LIN {X 0,Y 369.044,Z 241.011,A -85,B 0,C 180,E1 -12789.865,E2 -12789.865} C_VEL
LIN {X 0,Y 369.022,Z 241.014,A -85,B 0,C 180,E1 -12793.768,E2 -12793.768} C_VEL
LIN {X 0,Y 368.974,Z 241.02,A -85,B 0,C 180,E1 -12797.739,E2 -12797.739} C_VEL
LIN {X 0,Y 368.891,Z 241.032,A -85,B 0,C 180,E1 -12801.217,E2 -12801.217} C_VEL
LIN {X 0,Y 368.912,Z 241.029,A -85,B 0,C 180,E1 -12804.774,E2 -12804.774} C_VEL
LIN {X 0,Y 368.894,Z 241.025,A -85,B 0,C 180,E1 -12808.438,E2 -12808.438} C_VEL
LIN {X 0,Y 368.874,Z 241.03,A -85,B 0,C 180,E1 -12812.235,E2 -12812.235} C_VEL
LIN {X 0,Y 368.905,Z 241.028,A -85,B 0,C 180,E1 -12814.998,E2 -12814.998} C_VEL
LIN {X 0,Y 368.887,Z 241.036,A -85,B 0,C 180,E1 -12818.638,E2 -12818.638} C_VEL
LIN {X 0,Y 368.952,Z 241.097,A -85,B 0,C 180,E1 -12820.366,E2 -12820.366} C_VEL
LIN {X 0,Y 370.279,Z 247.105,A -85,B 0,C 180,E1 -12822.072,E2 -12822.072} C_VEL
LIN {X 0,Y 372.182,Z 257.131,A -85,B 0,C 180,E1 -12824.693,E2 -12824.693} C_VEL
LIN {X 0,Y 372.185,Z 259.385,A -85,B 0,C 180,E1 -12825.156,E2 -12825.156} C_VEL
LIN {X 0,Y 376.972,Z 282.842,A -85,B 0,C 180,E1 -12825.983,E2 -12825.983} C_VEL
LIN {X 0,Y 377.58,Z 287.336,A -85,B 0,C 180,E1 -12826.115,E2 -12826.115} C_VEL
LIN {X 0,Y 376.049,Z 367.06,A -85,B 0,C 180,E1 -12827.695,E2 -12827.695} C_VEL
LIN {X 0,Y 375.45,Z 380.427,A -85,B 0,C 180,E1 -12828.176,E2 -12828.176} C_VEL
LIN {X 0,Y 374.723,Z 393.48,A -85,B 0,C 180,E1 -12828.884,E2 -12828.884} C_VEL
LIN {X 0,Y 373.829,Z 405.095,A -85,B 0,C 180,E1 -12829.742,E2 -12829.742} C_VEL
LIN {X 0,Y 372.648,Z 417.198,A -85,B 0,C 180,E1 -12830.894,E2 -12830.894} C_VEL
LIN {X 0,Y 371.644,Z 427.056,A -85,B 0,C 180,E1 -12832.08,E2 -12832.08} C_VEL
LIN {X 0,Y 370.718,Z 435.571,A -85,B 0,C 180,E1 -12833.334,E2 -12833.334} C_VEL
LIN {X 0,Y 369.704,Z 444.74,A -85,B 0,C 180,E1 -12835.006,E2 -12835.006} C_VEL
LIN {X 0,Y 368.986,Z 451.255,A -85,B 0,C 180,E1 -12836.473,E2 -12836.473} C_VEL
LIN {X 0,Y 368.284,Z 457.921,A -85,B 0,C 180,E1 -12838.348,E2 -12838.348} C_VEL
LIN {X 0,Y 367.826,Z 462.929,A -85,B 0,C 180,E1 -12840.214,E2 -12840.214} C_VEL
LIN {X 0,Y 367.579,Z 465.737,A -85,B 0,C 180,E1 -12841.571,E2 -12841.571} C_VEL
LIN {X 0,Y 367.38,Z 467.49,A -85,B 0,C 180,E1 -12842.671,E2 -12842.671} C_VEL
LIN {X 0,Y 367.234,Z 469.127,A -85,B 0,C 180,E1 -12844.076,E2 -12844.076} C_VEL
LIN {X 0,Y 367.144,Z 469.909,A -85,B 0,C 180,E1 -12845.095,E2 -12845.095} C_VEL
LIN {X 0,Y 367.118,Z 470.416,A -85,B 0,C 180,E1 -12846.752,E2 -12846.752} C_VEL
LIN {X 0,Y 367.121,Z 469.889,A -85,B 0,C 180,E1 -12848.672,E2 -12848.672} C_VEL
LIN {X 0,Y 367.223,Z 468.929,A -85,B 0,C 180,E1 -12849.851,E2 -12849.851} C_VEL
LIN {X 0,Y 367.326,Z 467.538,A -85,B 0,C 180,E1 -12851.02,E2 -12851.02} C_VEL
LIN {X 0,Y 367.596,Z 464.278,A -85,B 0,C 180,E1 -12852.91,E2 -12852.91} C_VEL
LIN {X 0,Y 367.867,Z 460.491,A -85,B 0,C 180,E1 -12854.488,E2 -12854.488} C_VEL
LIN {X 0,Y 368.367,Z 455.285,A -85,B 0,C 180,E1 -12856.176,E2 -12856.176} C_VEL
LIN {X 0,Y 368.997,Z 448.471,A -85,B 0,C 180,E1 -12857.908,E2 -12857.908} C_VEL
LIN {X 0,Y 369.827,Z 440.094,A -85,B 0,C 180,E1 -12859.6,E2 -12859.6} C_VEL
LIN {X 0,Y 370.758,Z 430.811,A -85,B 0,C 180,E1 -12861.106,E2 -12861.106} C_VEL
LIN {X 0,Y 371.714,Z 420.895,A -85,B 0,C 180,E1 -12862.396,E2 -12862.396} C_VEL
LIN {X 0,Y 372.696,Z 410.311,A -85,B 0,C 180,E1 -12863.504,E2 -12863.504} C_VEL
LIN {X 0,Y 373.641,Z 398.688,A -85,B 0,C 180,E1 -12864.469,E2 -12864.469} C_VEL
LIN {X 0,Y 374.319,Z 386.768,A -85,B 0,C 180,E1 -12865.222,E2 -12865.222} C_VEL
LIN {X 0,Y 375.026,Z 373.695,A -85,B 0,C 180,E1 -12865.803,E2 -12865.803} C_VEL
LIN {X 0,Y 375.431,Z 360.14,A -85,B 0,C 180,E1 -12866.177,E2 -12866.177} C_VEL
LIN {X 0,Y 376.575,Z 285.809,A -85,B 0,C 180,E1 -12867.62,E2 -12867.62} C_VEL
LIN {X 0,Y 371.712,Z 259.806,A -85,B 0,C 180,E1 -12868.444,E2 -12868.444} C_VEL
LIN {X 0,Y 371.685,Z 258.504,A -85,B 0,C 180,E1 -12868.647,E2 -12868.647} C_VEL
LIN {X 0,Y 371.677,Z 254.292,A -85,B 0,C 180,E1 -12869.73,E2 -12869.73} C_VEL
LIN {X 0,Y 370.534,Z 247.731,A -85,B 0,C 180,E1 -12871.523,E2 -12871.523} C_VEL
LIN {X 0,Y 369.47,Z 246.002,A -85,B 0,C 180,E1 -12872.056,E2 -12872.056} C_VEL
LIN {X 0,Y 366.012,Z 243.763,A -85,B 0,C 180,E1 -12872.906,E2 -12872.906} C_VEL
LIN {X 0,Y 362.72,Z 242.239,A -85,B 0,C 180,E1 -12873.814,E2 -12873.814} C_VEL
LIN {X 0,Y 361.924,Z 241.9,A -85,B 0,C 180,E1 -12874.431,E2 -12874.431} C_VEL
LIN {X 0,Y 362.127,Z 241.873,A -85,B 0,C 180,E1 -12876.688,E2 -12876.688} C_VEL
LIN {X 0,Y 361.999,Z 241.891,A -85,B 0,C 180,E1 -12880.064,E2 -12880.064} C_VEL
LIN {X 0,Y 361.965,Z 241.895,A -85,B 0,C 180,E1 -12883.901,E2 -12883.901} C_VEL
LIN {X 0,Y 361.935,Z 241.904,A -85,B 0,C 180,E1 -12887.941,E2 -12887.941} C_VEL
LIN {X 0,Y 361.823,Z 241.914,A -85,B 0,C 180,E1 -12891.658,E2 -12891.658} C_VEL
LIN {X 0,Y 361.858,Z 241.905,A -85,B 0,C 180,E1 -12895.296,E2 -12895.296} C_VEL
LIN {X 0,Y 361.827,Z 241.901,A -85,B 0,C 180,E1 -12899.077,E2 -12899.077} C_VEL
LIN {X 0,Y 361.819,Z 241.911,A -85,B 0,C 180,E1 -12902.949,E2 -12902.949} C_VEL
LIN {X 0,Y 361.837,Z 241.897,A -85,B 0,C 180,E1 -12905.641,E2 -12905.641} C_VEL
LIN {X 0,Y 361.8,Z 241.916,A -85,B 0,C 180,E1 -12909.021,E2 -12909.021} C_VEL
LIN {X 0,Y 361.806,Z 241.902,A -85,B 0,C 180,E1 -12912.834,E2 -12912.834} C_VEL
LIN {X 0,Y 361.792,Z 241.915,A -85,B 0,C 180,E1 -12915.952,E2 -12915.952} C_VEL
LIN {X 0,Y 361.791,Z 241.907,A -85,B 0,C 180,E1 -12919.254,E2 -12919.254} C_VEL
LIN {X 0,Y 361.845,Z 241.898,A -85,B 0,C 180,E1 -12922.986,E2 -12922.986} C_VEL
LIN {X 0,Y 361.843,Z 241.911,A -85,B 0,C 180,E1 -12926.636,E2 -12926.636} C_VEL
LIN {X 0,Y 361.834,Z 241.894,A -85,B 0,C 180,E1 -12929.674,E2 -12929.674} C_VEL
LIN {X 0,Y 361.844,Z 241.899,A -85,B 0,C 180,E1 -12933.472,E2 -12933.472} C_VEL
LIN {X 0,Y 361.865,Z 241.909,A -85,B 0,C 180,E1 -12937.148,E2 -12937.148} C_VEL
LIN {X 0,Y 361.897,Z 241.888,A -85,B 0,C 180,E1 -12940.728,E2 -12940.728} C_VEL
LIN {X 0,Y 361.938,Z 241.884,A -85,B 0,C 180,E1 -12944.23,E2 -12944.23} C_VEL
LIN {X 0,Y 361.995,Z 241.887,A -85,B 0,C 180,E1 -12946.532,E2 -12946.532} C_VEL
LIN {X 0,Y 361.993,Z 241.889,A -85,B 0,C 180,E1 -12949.941,E2 -12949.941} C_VEL
LIN {X 0,Y 362.118,Z 241.853,A -85,B 0,C 180,E1 -12953.317,E2 -12953.317} C_VEL
LIN {X 0,Y 362.266,Z 241.852,A -85,B 0,C 180,E1 -12957.78,E2 -12957.78} C_VEL
LIN {X 0,Y 362.202,Z 241.861,A -85,B 0,C 180,E1 -12961.116,E2 -12961.116} C_VEL
LIN {X 0,Y 362.261,Z 241.852,A -85,B 0,C 180,E1 -12962.227,E2 -12962.227} C_VEL
LIN {X 0,Y 362.145,Z 241.857,A -85,B 0,C 180,E1 -12966.69,E2 -12966.69} C_VEL
LIN {X 0,Y 362.004,Z 241.89,A -85,B 0,C 180,E1 -12970.066,E2 -12970.066} C_VEL
LIN {X 0,Y 362.006,Z 241.879,A -85,B 0,C 180,E1 -12973.902,E2 -12973.902} C_VEL
LIN {X 0,Y 361.936,Z 241.889,A -85,B 0,C 180,E1 -12976.937,E2 -12976.937} C_VEL
LIN {X 0,Y 361.896,Z 241.906,A -85,B 0,C 180,E1 -12980.464,E2 -12980.464} C_VEL
LIN {X 0,Y 361.904,Z 241.882,A -85,B 0,C 180,E1 -12984.115,E2 -12984.115} C_VEL
LIN {X 0,Y 361.853,Z 241.909,A -85,B 0,C 180,E1 -12987.787,E2 -12987.787} C_VEL
LIN {X 0,Y 361.858,Z 241.899,A -85,B 0,C 180,E1 -12991.287,E2 -12991.287} C_VEL
LIN {X 0,Y 361.865,Z 241.907,A -85,B 0,C 180,E1 -12994.282,E2 -12994.282} C_VEL
LIN {X 0,Y 361.871,Z 241.901,A -85,B 0,C 180,E1 -12997.224,E2 -12997.224} C_VEL
LIN {X 0,Y 361.825,Z 241.912,A -85,B 0,C 180,E1 -13000.752,E2 -13000.752} C_VEL
LIN {X 0,Y 361.826,Z 241.913,A -85,B 0,C 180,E1 -13004.37,E2 -13004.37} C_VEL
LIN {X 0,Y 361.842,Z 241.912,A -85,B 0,C 180,E1 -13007.571,E2 -13007.571} C_VEL
LIN {X 0,Y 361.855,Z 241.911,A -85,B 0,C 180,E1 -13011.573,E2 -13011.573} C_VEL
LIN {X 0,Y 361.887,Z 241.907,A -85,B 0,C 180,E1 -13014.656,E2 -13014.656} C_VEL
LIN {X 0,Y 361.851,Z 241.913,A -85,B 0,C 180,E1 -13018.371,E2 -13018.371} C_VEL
LIN {X 0,Y 361.94,Z 241.978,A -85,B 0,C 180,E1 -13021.196,E2 -13021.196} C_VEL
LIN {X 0,Y 363.7,Z 250.571,A -85,B 0,C 180,E1 -13023.611,E2 -13023.611} C_VEL
LIN {X 0,Y 365.297,Z 259.104,A -85,B 0,C 180,E1 -13025.868,E2 -13025.868} C_VEL
LIN {X 0,Y 364.796,Z 266.345,A -85,B 0,C 180,E1 -13027.635,E2 -13027.635} C_VEL
LIN {X 0,Y 364.608,Z 268.699,A -85,B 0,C 180,E1 -13028.152,E2 -13028.152} C_VEL
LIN {X 0,Y 365.93,Z 276.421,A -85,B 0,C 180,E1 -13028.437,E2 -13028.437} C_VEL
LIN {X 0,Y 369.774,Z 299.232,A -85,B 0,C 180,E1 -13029.125,E2 -13029.125} C_VEL
LIN {X 0,Y 368.476,Z 376.627,A -85,B 0,C 180,E1 -13030.682,E2 -13030.682} C_VEL
LIN {X 0,Y 367.861,Z 389.768,A -85,B 0,C 180,E1 -13031.155,E2 -13031.155} C_VEL
LIN {X 0,Y 367.089,Z 401.886,A -85,B 0,C 180,E1 -13031.801,E2 -13031.801} C_VEL
LIN {X 0,Y 366.077,Z 414.134,A -85,B 0,C 180,E1 -13032.687,E2 -13032.687} C_VEL
LIN {X 0,Y 365.009,Z 425.73,A -85,B 0,C 180,E1 -13033.787,E2 -13033.787} C_VEL
LIN {X 0,Y 364.045,Z 436.165,A -85,B 0,C 180,E1 -13035.034,E2 -13035.034} C_VEL
LIN {X 0,Y 363.234,Z 444.713,A -85,B 0,C 180,E1 -13036.289,E2 -13036.289} C_VEL
LIN {X 0,Y 362.169,Z 453.947,A -85,B 0,C 180,E1 -13037.958,E2 -13037.958} C_VEL
LIN {X 0,Y 361.457,Z 461.37,A -85,B 0,C 180,E1 -13039.638,E2 -13039.638} C_VEL
LIN {X 0,Y 360.855,Z 468.19,A -85,B 0,C 180,E1 -13041.6,E2 -13041.6} C_VEL
LIN {X 0,Y 360.52,Z 472.681,A -85,B 0,C 180,E1 -13043.282,E2 -13043.282} C_VEL
LIN {X 0,Y 360.409,Z 475.047,A -85,B 0,C 180,E1 -13044.404,E2 -13044.404} C_VEL
LIN {X 0,Y 360.355,Z 476.982,A -85,B 0,C 180,E1 -13045.525,E2 -13045.525} C_VEL
LIN {X 0,Y 360.279,Z 478.488,A -85,B 0,C 180,E1 -13046.644,E2 -13046.644} C_VEL
LIN {X 0,Y 360.254,Z 480.203,A -85,B 0,C 180,E1 -13048.881,E2 -13048.881} C_VEL
LIN {X 0,Y 360.28,Z 480.477,A -85,B 0,C 180,E1 -13049.999,E2 -13049.999} C_VEL
LIN {X 0,Y 360.253,Z 480.354,A -85,B 0,C 180,E1 -13051.117,E2 -13051.117} C_VEL
LIN {X 0,Y 360.282,Z 478.849,A -85,B 0,C 180,E1 -13053.354,E2 -13053.354} C_VEL
LIN {X 0,Y 360.383,Z 477.507,A -85,B 0,C 180,E1 -13054.473,E2 -13054.473} C_VEL
LIN {X 0,Y 360.47,Z 474.804,A -85,B 0,C 180,E1 -13056.084,E2 -13056.084} C_VEL
LIN {X 0,Y 360.757,Z 470.803,A -85,B 0,C 180,E1 -13057.837,E2 -13057.837} C_VEL
LIN {X 0,Y 361.229,Z 465.814,A -85,B 0,C 180,E1 -13059.518,E2 -13059.518} C_VEL
LIN {X 0,Y 361.887,Z 459.549,A -85,B 0,C 180,E1 -13061.197,E2 -13061.197} C_VEL
LIN {X 0,Y 362.802,Z 451.718,A -85,B 0,C 180,E1 -13062.871,E2 -13062.871} C_VEL
LIN {X 0,Y 363.967,Z 441.947,A -85,B 0,C 180,E1 -13064.537,E2 -13064.537} C_VEL
LIN {X 0,Y 364.975,Z 431.82,A -85,B 0,C 180,E1 -13065.925,E2 -13065.925} C_VEL
LIN {X 0,Y 366.099,Z 421.791,A -85,B 0,C 180,E1 -13067.022,E2 -13067.022} C_VEL
LIN {X 0,Y 367.139,Z 410.901,A -85,B 0,C 180,E1 -13067.978,E2 -13067.978} C_VEL
LIN {X 0,Y 368.134,Z 398.889,A -85,B 0,C 180,E1 -13068.792,E2 -13068.792} C_VEL
LIN {X 0,Y 368.934,Z 386.604,A -85,B 0,C 180,E1 -13069.4,E2 -13069.4} C_VEL
LIN {X 0,Y 369.469,Z 374.043,A -85,B 0,C 180,E1 -13069.804,E2 -13069.804} C_VEL
LIN {X 0,Y 370.794,Z 299.844,A -85,B 0,C 180,E1 -13071.297,E2 -13071.297} C_VEL
LIN {X 0,Y 366.754,Z 276.745,A -85,B 0,C 180,E1 -13072.058,E2 -13072.058} C_VEL
LIN {X 0,Y 365.053,Z 268.304,A -85,B 0,C 180,E1 -13072.397,E2 -13072.397} C_VEL
LIN {X 0,Y 365.707,Z 260.961,A -85,B 0,C 180,E1 -13074.101,E2 -13074.101} C_VEL
LIN {X 0,Y 363.888,Z 250.827,A -85,B 0,C 180,E1 -13076.78,E2 -13076.78} C_VEL
LIN {X 0,Y 361.943,Z 242.234,A -85,B 0,C 180,E1 -13079.183,E2 -13079.183} C_VEL
LIN {X 0,Y 361.888,Z 241.905,A -85,B 0,C 180,E1 -13079.682,E2 -13079.682} C_VEL
LIN {X 0,Y 361.865,Z 241.908,A -85,B 0,C 180,E1 -13083.367,E2 -13083.367} C_VEL
LIN {X 0,Y 361.869,Z 241.902,A -85,B 0,C 180,E1 -13087.016,E2 -13087.016} C_VEL
LIN {X 0,Y 361.818,Z 241.908,A -85,B 0,C 180,E1 -13090.749,E2 -13090.749} C_VEL
LIN {X 0,Y 361.821,Z 241.918,A -85,B 0,C 180,E1 -13094.366,E2 -13094.366} C_VEL
LIN {X 0,Y 361.834,Z 241.912,A -85,B 0,C 180,E1 -13097.567,E2 -13097.567} C_VEL
LIN {X 0,Y 361.845,Z 241.905,A -85,B 0,C 180,E1 -13101.569,E2 -13101.569} C_VEL
LIN {X 0,Y 361.872,Z 241.905,A -85,B 0,C 180,E1 -13104.653,E2 -13104.653} C_VEL
LIN {X 0,Y 361.839,Z 241.908,A -85,B 0,C 180,E1 -13108.367,E2 -13108.367} C_VEL
LIN {X 0,Y 361.867,Z 241.909,A -85,B 0,C 180,E1 -13110.949,E2 -13110.949} C_VEL
LIN {X 0,Y 361.879,Z 241.909,A -85,B 0,C 180,E1 -13114.703,E2 -13114.703} C_VEL
LIN {X 0,Y 361.859,Z 241.905,A -85,B 0,C 180,E1 -13118.342,E2 -13118.342} C_VEL
LIN {X 0,Y 361.918,Z 241.892,A -85,B 0,C 180,E1 -13122.081,E2 -13122.081} C_VEL
LIN {X 0,Y 361.958,Z 241.893,A -85,B 0,C 180,E1 -13125.376,E2 -13125.376} C_VEL
LIN {X 0,Y 361.962,Z 241.896,A -85,B 0,C 180,E1 -13128.801,E2 -13128.801} C_VEL
LIN {X 0,Y 362.08,Z 241.876,A -85,B 0,C 180,E1 -13132.187,E2 -13132.187} C_VEL
LIN {X 0,Y 362.092,Z 241.879,A -85,B 0,C 180,E1 -13134.427,E2 -13134.427} C_VEL
LIN {X 0,Y 362.248,Z 241.861,A -85,B 0,C 180,E1 -13137.773,E2 -13137.773} C_VEL
LIN {X 0,Y 362.245,Z 241.86,A -85,B 0,C 180,E1 -13142.22,E2 -13142.22} C_VEL
LIN {X 0,Y 362.103,Z 241.876,A -85,B 0,C 180,E1 -13146.683,E2 -13146.683} C_VEL
LIN {X 0,Y 361.981,Z 241.891,A -85,B 0,C 180,E1 -13150.059,E2 -13150.059} C_VEL
LIN {X 0,Y 361.983,Z 241.891,A -85,B 0,C 180,E1 -13153.895,E2 -13153.895} C_VEL
LIN {X 0,Y 361.911,Z 241.897,A -85,B 0,C 180,E1 -13156.93,E2 -13156.93} C_VEL
LIN {X 0,Y 361.868,Z 241.908,A -85,B 0,C 180,E1 -13160.457,E2 -13160.457} C_VEL
LIN {X 0,Y 361.874,Z 241.91,A -85,B 0,C 180,E1 -13164.109,E2 -13164.109} C_VEL
LIN {X 0,Y 361.826,Z 241.911,A -85,B 0,C 180,E1 -13167.781,E2 -13167.781} C_VEL
LIN {X 0,Y 361.824,Z 241.912,A -85,B 0,C 180,E1 -13171.282,E2 -13171.282} C_VEL
LIN {X 0,Y 361.83,Z 241.914,A -85,B 0,C 180,E1 -13174.277,E2 -13174.277} C_VEL
LIN {X 0,Y 361.84,Z 241.909,A -85,B 0,C 180,E1 -13177.22,E2 -13177.22} C_VEL
LIN {X 0,Y 361.887,Z 242.014,A -85,B 0,C 180,E1 -13179.991,E2 -13179.991} C_VEL
LIN {X 0,Y 364.059,Z 252.05,A -85,B 0,C 180,E1 -13182.815,E2 -13182.815} C_VEL
LIN {X 0,Y 365.336,Z 259.235,A -85,B 0,C 180,E1 -13184.666,E2 -13184.666} C_VEL
LIN {X 0,Y 367.968,Z 271.225,A -85,B 0,C 180,E1 -13185.148,E2 -13185.148} C_VEL
LIN {X 0,Y 371.016,Z 287.413,A -85,B 0,C 180,E1 -13185.696,E2 -13185.696} C_VEL
LIN {X 0,Y 369.417,Z 367.303,A -85,B 0,C 180,E1 -13187.311,E2 -13187.311} C_VEL
LIN {X 0,Y 368.798,Z 380.614,A -85,B 0,C 180,E1 -13187.801,E2 -13187.801} C_VEL
LIN {X 0,Y 368.035,Z 393.611,A -85,B 0,C 180,E1 -13188.519,E2 -13188.519} C_VEL
LIN {X 0,Y 367.098,Z 405.197,A -85,B 0,C 180,E1 -13189.39,E2 -13189.39} C_VEL
LIN {X 0,Y 365.995,Z 416.282,A -85,B 0,C 180,E1 -13190.456,E2 -13190.456} C_VEL
LIN {X 0,Y 364.811,Z 427.131,A -85,B 0,C 180,E1 -13191.767,E2 -13191.767} C_VEL
LIN {X 0,Y 363.731,Z 436.589,A -85,B 0,C 180,E1 -13193.205,E2 -13193.205} C_VEL
LIN {X 0,Y 362.748,Z 445.105,A -85,B 0,C 180,E1 -13194.805,E2 -13194.805} C_VEL
LIN {X 0,Y 362.014,Z 451.36,A -85,B 0,C 180,E1 -13196.245,E2 -13196.245} C_VEL
LIN {X 0,Y 361.421,Z 456.486,A -85,B 0,C 180,E1 -13197.674,E2 -13197.674} C_VEL
LIN {X 0,Y 360.904,Z 461.912,A -85,B 0,C 180,E1 -13199.583,E2 -13199.583} C_VEL
LIN {X 0,Y 360.531,Z 465.562,A -85,B 0,C 180,E1 -13201.295,E2 -13201.295} C_VEL
LIN {X 0,Y 360.212,Z 468.571,A -85,B 0,C 180,E1 -13203.338,E2 -13203.338} C_VEL
LIN {X 0,Y 360.091,Z 469.685,A -85,B 0,C 180,E1 -13204.573,E2 -13204.573} C_VEL
LIN {X 0,Y 360.012,Z 470.491,A -85,B 0,C 180,E1 -13206.551,E2 -13206.551} C_VEL
LIN {X 0,Y 360.028,Z 470.193,A -85,B 0,C 180,E1 -13208.23,E2 -13208.23} C_VEL
LIN {X 0,Y 360.1,Z 469.392,A -85,B 0,C 180,E1 -13209.506,E2 -13209.506} C_VEL
LIN {X 0,Y 360.201,Z 468.215,A -85,B 0,C 180,E1 -13210.63,E2 -13210.63} C_VEL
LIN {X 0,Y 360.482,Z 464.784,A -85,B 0,C 180,E1 -13212.787,E2 -13212.787} C_VEL
LIN {X 0,Y 360.852,Z 460.199,A -85,B 0,C 180,E1 -13214.757,E2 -13214.757} C_VEL
LIN {X 0,Y 361.381,Z 454.762,A -85,B 0,C 180,E1 -13216.505,E2 -13216.505} C_VEL
LIN {X 0,Y 362.03,Z 447.928,A -85,B 0,C 180,E1 -13218.24,E2 -13218.24} C_VEL
LIN {X 0,Y 362.962,Z 439.404,A -85,B 0,C 180,E1 -13219.965,E2 -13219.965} C_VEL
LIN {X 0,Y 363.867,Z 430.631,A -85,B 0,C 180,E1 -13221.392,E2 -13221.392} C_VEL
LIN {X 0,Y 364.97,Z 419.749,A -85,B 0,C 180,E1 -13222.811,E2 -13222.811} C_VEL
LIN {X 0,Y 366,Z 408.903,A -85,B 0,C 180,E1 -13223.939,E2 -13223.939} C_VEL
LIN {X 0,Y 366.903,Z 397.811,A -85,B 0,C 180,E1 -13224.846,E2 -13224.846} C_VEL
LIN {X 0,Y 367.615,Z 385.485,A -85,B 0,C 180,E1 -13225.615,E2 -13225.615} C_VEL
LIN {X 0,Y 368.272,Z 372.83,A -85,B 0,C 180,E1 -13226.171,E2 -13226.171} C_VEL
LIN {X 0,Y 368.693,Z 360.056,A -85,B 0,C 180,E1 -13226.518,E2 -13226.518} C_VEL
LIN {X 0,Y 369.847,Z 286.54,A -85,B 0,C 180,E1 -13227.973,E2 -13227.973} C_VEL
LIN {X 0,Y 364.875,Z 260.049,A -85,B 0,C 180,E1 -13228.829,E2 -13228.829} C_VEL
LIN {X 0,Y 364.799,Z 258.971,A -85,B 0,C 180,E1 -13228.966,E2 -13228.966} C_VEL
LIN {X 0,Y 364.641,Z 255.007,A -85,B 0,C 180,E1 -13230.001,E2 -13230.001} C_VEL
LIN {X 0,Y 362.806,Z 245.13,A -85,B 0,C 180,E1 -13232.777,E2 -13232.777} C_VEL
LIN {X 0,Y 361.995,Z 241.924,A -85,B 0,C 180,E1 -13233.793,E2 -13233.793} C_VEL
LIN {X 0,Y 361.924,Z 241.9,A -85,B 0,C 180,E1 -13234.431,E2 -13234.431} C_VEL
LIN {X 0,Y 361.258,Z 241.986,A -85,B 0,C 180,E1 -13235.36,E2 -13235.36} C_VEL
LIN {X 0,Y 358.461,Z 242.33,A -85,B 0,C 180,E1 -13236.874,E2 -13236.874} C_VEL
LIN {X 0,Y 356.086,Z 242.63,A -85,B 0,C 180,E1 -13238.098,E2 -13238.098} C_VEL
LIN {X 0,Y 355.048,Z 242.755,A -85,B 0,C 180,E1 -13239.044,E2 -13239.044} C_VEL
LIN {X 0,Y 354.953,Z 242.765,A -85,B 0,C 180,E1 -13239.365,E2 -13239.365} C_VEL
LIN {X 0,Y 354.891,Z 242.767,A -85,B 0,C 180,E1 -13242.583,E2 -13242.583} C_VEL
LIN {X 0,Y 354.856,Z 242.778,A -85,B 0,C 180,E1 -13246.098,E2 -13246.098} C_VEL
LIN {X 0,Y 354.869,Z 242.779,A -85,B 0,C 180,E1 -13248.475,E2 -13248.475} C_VEL
LIN {X 0,Y 354.777,Z 242.794,A -85,B 0,C 180,E1 -13252.111,E2 -13252.111} C_VEL
LIN {X 0,Y 354.82,Z 242.782,A -85,B 0,C 180,E1 -13254.58,E2 -13254.58} C_VEL
LIN {X 0,Y 354.773,Z 242.784,A -85,B 0,C 180,E1 -13258.389,E2 -13258.389} C_VEL
LIN {X 0,Y 354.757,Z 242.797,A -85,B 0,C 180,E1 -13262.337,E2 -13262.337} C_VEL
LIN {X 0,Y 354.792,Z 242.775,A -85,B 0,C 180,E1 -13265.702,E2 -13265.702} C_VEL
LIN {X 0,Y 354.744,Z 242.794,A -85,B 0,C 180,E1 -13269.416,E2 -13269.416} C_VEL
LIN {X 0,Y 354.758,Z 242.779,A -85,B 0,C 180,E1 -13272.87,E2 -13272.87} C_VEL
LIN {X 0,Y 354.741,Z 242.794,A -85,B 0,C 180,E1 -13276.107,E2 -13276.107} C_VEL
LIN {X 0,Y 354.743,Z 242.785,A -85,B 0,C 180,E1 -13279.18,E2 -13279.18} C_VEL
LIN {X 0,Y 354.782,Z 242.772,A -85,B 0,C 180,E1 -13282.409,E2 -13282.409} C_VEL
LIN {X 0,Y 354.792,Z 242.788,A -85,B 0,C 180,E1 -13284.945,E2 -13284.945} C_VEL
LIN {X 0,Y 354.779,Z 242.784,A -85,B 0,C 180,E1 -13288.41,E2 -13288.41} C_VEL
LIN {X 0,Y 354.777,Z 242.766,A -85,B 0,C 180,E1 -13291.618,E2 -13291.618} C_VEL
LIN {X 0,Y 354.796,Z 242.788,A -85,B 0,C 180,E1 -13295.424,E2 -13295.424} C_VEL
LIN {X 0,Y 354.819,Z 242.783,A -85,B 0,C 180,E1 -13299.118,E2 -13299.118} C_VEL
LIN {X 0,Y 354.874,Z 242.746,A -85,B 0,C 180,E1 -13302.723,E2 -13302.723} C_VEL
LIN {X 0,Y 354.948,Z 242.767,A -85,B 0,C 180,E1 -13306.259,E2 -13306.259} C_VEL
LIN {X 0,Y 354.949,Z 242.769,A -85,B 0,C 180,E1 -13309.739,E2 -13309.739} C_VEL
LIN {X 0,Y 355.084,Z 242.729,A -85,B 0,C 180,E1 -13313.184,E2 -13313.184} C_VEL
LIN {X 0,Y 355.228,Z 242.728,A -85,B 0,C 180,E1 -13317.736,E2 -13317.736} C_VEL
LIN {X 0,Y 355.171,Z 242.737,A -85,B 0,C 180,E1 -13321.138,E2 -13321.138} C_VEL
LIN {X 0,Y 355.223,Z 242.727,A -85,B 0,C 180,E1 -13322.272,E2 -13322.272} C_VEL
LIN {X 0,Y 355.109,Z 242.735,A -85,B 0,C 180,E1 -13326.823,E2 -13326.823} C_VEL
LIN {X 0,Y 354.96,Z 242.77,A -85,B 0,C 180,E1 -13330.268,E2 -13330.268} C_VEL
LIN {X 0,Y 354.951,Z 242.758,A -85,B 0,C 180,E1 -13334.022,E2 -13334.022} C_VEL
LIN {X 0,Y 354.899,Z 242.77,A -85,B 0,C 180,E1 -13338.095,E2 -13338.095} C_VEL
LIN {X 0,Y 354.825,Z 242.78,A -85,B 0,C 180,E1 -13342.11,E2 -13342.11} C_VEL
LIN {X 0,Y 354.859,Z 242.762,A -85,B 0,C 180,E1 -13344.58,E2 -13344.58} C_VEL
LIN {X 0,Y 354.811,Z 242.786,A -85,B 0,C 180,E1 -13348.388,E2 -13348.388} C_VEL
LIN {X 0,Y 354.798,Z 242.78,A -85,B 0,C 180,E1 -13352.336,E2 -13352.336} C_VEL
LIN {X 0,Y 354.833,Z 242.782,A -85,B 0,C 180,E1 -13355.701,E2 -13355.701} C_VEL
LIN {X 0,Y 354.78,Z 242.792,A -85,B 0,C 180,E1 -13359.414,E2 -13359.414} C_VEL
LIN {X 0,Y 354.797,Z 242.779,A -85,B 0,C 180,E1 -13362.868,E2 -13362.868} C_VEL
LIN {X 0,Y 354.775,Z 242.788,A -85,B 0,C 180,E1 -13366.104,E2 -13366.104} C_VEL
LIN {X 0,Y 354.778,Z 242.791,A -85,B 0,C 180,E1 -13369.177,E2 -13369.177} C_VEL
LIN {X 0,Y 354.813,Z 242.789,A -85,B 0,C 180,E1 -13372.405,E2 -13372.405} C_VEL
LIN {X 0,Y 354.825,Z 242.786,A -85,B 0,C 180,E1 -13374.941,E2 -13374.941} C_VEL
LIN {X 0,Y 354.807,Z 242.79,A -85,B 0,C 180,E1 -13378.406,E2 -13378.406} C_VEL
LIN {X 0,Y 354.912,Z 242.982,A -85,B 0,C 180,E1 -13380.945,E2 -13380.945} C_VEL
LIN {X 0,Y 356.904,Z 252.771,A -85,B 0,C 180,E1 -13383.7,E2 -13383.7} C_VEL
LIN {X 0,Y 358.388,Z 261.296,A -85,B 0,C 180,E1 -13385.988,E2 -13385.988} C_VEL
LIN {X 0,Y 357.76,Z 268.482,A -85,B 0,C 180,E1 -13387.722,E2 -13387.722} C_VEL
LIN {X 0,Y 358.319,Z 272.203,A -85,B 0,C 180,E1 -13387.904,E2 -13387.904} C_VEL
LIN {X 0,Y 363.103,Z 300.432,A -85,B 0,C 180,E1 -13388.78,E2 -13388.78} C_VEL
LIN {X 0,Y 361.716,Z 376.81,A -85,B 0,C 180,E1 -13390.343,E2 -13390.343} C_VEL
LIN {X 0,Y 361.088,Z 389.856,A -85,B 0,C 180,E1 -13390.825,E2 -13390.825} C_VEL
LIN {X 0,Y 360.243,Z 402.49,A -85,B 0,C 180,E1 -13391.516,E2 -13391.516} C_VEL
LIN {X 0,Y 359.278,Z 413.736,A -85,B 0,C 180,E1 -13392.349,E2 -13392.349} C_VEL
LIN {X 0,Y 358.188,Z 425.388,A -85,B 0,C 180,E1 -13393.47,E2 -13393.47} C_VEL
LIN {X 0,Y 357.123,Z 435.864,A -85,B 0,C 180,E1 -13394.737,E2 -13394.737} C_VEL
LIN {X 0,Y 356.286,Z 444.446,A -85,B 0,C 180,E1 -13396.016,E2 -13396.016} C_VEL
LIN {X 0,Y 355.382,Z 452.343,A -85,B 0,C 180,E1 -13397.435,E2 -13397.435} C_VEL
LIN {X 0,Y 354.574,Z 460.045,A -85,B 0,C 180,E1 -13399.146,E2 -13399.146} C_VEL
LIN {X 0,Y 353.98,Z 466.229,A -85,B 0,C 180,E1 -13400.86,E2 -13400.86} C_VEL
LIN {X 0,Y 353.543,Z 471.132,A -85,B 0,C 180,E1 -13402.575,E2 -13402.575} C_VEL
LIN {X 0,Y 353.341,Z 474.902,A -85,B 0,C 180,E1 -13404.292,E2 -13404.292} C_VEL
LIN {X 0,Y 353.271,Z 476.844,A -85,B 0,C 180,E1 -13405.435,E2 -13405.435} C_VEL
LIN {X 0,Y 353.203,Z 478.363,A -85,B 0,C 180,E1 -13406.577,E2 -13406.577} C_VEL
LIN {X 0,Y 353.154,Z 480.094,A -85,B 0,C 180,E1 -13408.859,E2 -13408.859} C_VEL
LIN {X 0,Y 353.181,Z 480.375,A -85,B 0,C 180,E1 -13409.999,E2 -13409.999} C_VEL
LIN {X 0,Y 353.153,Z 480.262,A -85,B 0,C 180,E1 -13411.139,E2 -13411.139} C_VEL
LIN {X 0,Y 353.208,Z 478.773,A -85,B 0,C 180,E1 -13413.421,E2 -13413.421} C_VEL
LIN {X 0,Y 353.299,Z 477.437,A -85,B 0,C 180,E1 -13414.563,E2 -13414.563} C_VEL
LIN {X 0,Y 353.398,Z 474.987,A -85,B 0,C 180,E1 -13416.078,E2 -13416.078} C_VEL
LIN {X 0,Y 353.712,Z 470.761,A -85,B 0,C 180,E1 -13417.994,E2 -13417.994} C_VEL
LIN {X 0,Y 354.19,Z 465.786,A -85,B 0,C 180,E1 -13419.709,E2 -13419.709} C_VEL
LIN {X 0,Y 354.884,Z 459.54,A -85,B 0,C 180,E1 -13421.421,E2 -13421.421} C_VEL
LIN {X 0,Y 355.877,Z 451.745,A -85,B 0,C 180,E1 -13423.126,E2 -13423.126} C_VEL
LIN {X 0,Y 357.081,Z 442.009,A -85,B 0,C 180,E1 -13424.824,E2 -13424.824} C_VEL
LIN {X 0,Y 358.154,Z 431.942,A -85,B 0,C 180,E1 -13426.237,E2 -13426.237} C_VEL
LIN {X 0,Y 359.435,Z 420.547,A -85,B 0,C 180,E1 -13427.494,E2 -13427.494} C_VEL
LIN {X 0,Y 360.592,Z 409.383,A -85,B 0,C 180,E1 -13428.463,E2 -13428.463} C_VEL
LIN {X 0,Y 361.542,Z 398.104,A -85,B 0,C 180,E1 -13429.222,E2 -13429.222} C_VEL
LIN {X 0,Y 362.367,Z 385.417,A -85,B 0,C 180,E1 -13429.84,E2 -13429.84} C_VEL
LIN {X 0,Y 362.922,Z 372.162,A -85,B 0,C 180,E1 -13430.251,E2 -13430.251} C_VEL
LIN {X 0,Y 364.264,Z 300.802,A -85,B 0,C 180,E1 -13431.706,E2 -13431.706} C_VEL
LIN {X 0,Y 360.329,Z 278.292,A -85,B 0,C 180,E1 -13432.471,E2 -13432.471} C_VEL
LIN {X 0,Y 358.317,Z 268.45,A -85,B 0,C 180,E1 -13432.856,E2 -13432.856} C_VEL
LIN {X 0,Y 358.509,Z 265.913,A -85,B 0,C 180,E1 -13433.388,E2 -13433.388} C_VEL
LIN {X 0,Y 358.794,Z 262.248,A -85,B 0,C 180,E1 -13434.288,E2 -13434.288} C_VEL
LIN {X 0,Y 356.763,Z 251.157,A -85,B 0,C 180,E1 -13437.291,E2 -13437.291} C_VEL
LIN {X 0,Y 354.864,Z 242.877,A -85,B 0,C 180,E1 -13439.717,E2 -13439.717} C_VEL
LIN {X 0,Y 354.814,Z 242.784,A -85,B 0,C 180,E1 -13443.7,E2 -13443.7} C_VEL
LIN {X 0,Y 354.801,Z 242.782,A -85,B 0,C 180,E1 -13446.458,E2 -13446.458} C_VEL
LIN {X 0,Y 354.774,Z 242.787,A -85,B 0,C 180,E1 -13449.41,E2 -13449.41} C_VEL
LIN {X 0,Y 354.79,Z 242.787,A -85,B 0,C 180,E1 -13452.864,E2 -13452.864} C_VEL
LIN {X 0,Y 354.77,Z 242.791,A -85,B 0,C 180,E1 -13456.101,E2 -13456.101} C_VEL
LIN {X 0,Y 354.769,Z 242.792,A -85,B 0,C 180,E1 -13459.173,E2 -13459.173} C_VEL
LIN {X 0,Y 354.802,Z 242.787,A -85,B 0,C 180,E1 -13462.402,E2 -13462.402} C_VEL
LIN {X 0,Y 354.81,Z 242.784,A -85,B 0,C 180,E1 -13464.937,E2 -13464.937} C_VEL
LIN {X 0,Y 354.794,Z 242.786,A -85,B 0,C 180,E1 -13468.402,E2 -13468.402} C_VEL
LIN {X 0,Y 354.797,Z 242.785,A -85,B 0,C 180,E1 -13471.611,E2 -13471.611} C_VEL
LIN {X 0,Y 354.834,Z 242.781,A -85,B 0,C 180,E1 -13475.654,E2 -13475.654} C_VEL
LIN {X 0,Y 354.825,Z 242.789,A -85,B 0,C 180,E1 -13479.11,E2 -13479.11} C_VEL
LIN {X 0,Y 354.878,Z 242.772,A -85,B 0,C 180,E1 -13482.715,E2 -13482.715} C_VEL
LIN {X 0,Y 354.948,Z 242.762,A -85,B 0,C 180,E1 -13486.252,E2 -13486.252} C_VEL
LIN {X 0,Y 354.948,Z 242.768,A -85,B 0,C 180,E1 -13489.731,E2 -13489.731} C_VEL
LIN {X 0,Y 355.097,Z 242.75,A -85,B 0,C 180,E1 -13493.176,E2 -13493.176} C_VEL
LIN {X 0,Y 355.21,Z 242.737,A -85,B 0,C 180,E1 -13497.728,E2 -13497.728} C_VEL
LIN {X 0,Y 355.134,Z 242.74,A -85,B 0,C 180,E1 -13501.13,E2 -13501.13} C_VEL
LIN {X 0,Y 355.207,Z 242.736,A -85,B 0,C 180,E1 -13502.264,E2 -13502.264} C_VEL
LIN {X 0,Y 355.07,Z 242.752,A -85,B 0,C 180,E1 -13506.816,E2 -13506.816} C_VEL
LIN {X 0,Y 354.937,Z 242.769,A -85,B 0,C 180,E1 -13510.261,E2 -13510.261} C_VEL
LIN {X 0,Y 354.928,Z 242.771,A -85,B 0,C 180,E1 -13514.015,E2 -13514.015} C_VEL
LIN {X 0,Y 354.873,Z 242.781,A -85,B 0,C 180,E1 -13518.088,E2 -13518.088} C_VEL
LIN {X 0,Y 354.8,Z 242.788,A -85,B 0,C 180,E1 -13521.414,E2 -13521.414} C_VEL
LIN {X 0,Y 354.831,Z 242.785,A -85,B 0,C 180,E1 -13524.573,E2 -13524.573} C_VEL
LIN {X 0,Y 354.78,Z 242.783,A -85,B 0,C 180,E1 -13528.382,E2 -13528.382} C_VEL
LIN {X 0,Y 354.763,Z 242.788,A -85,B 0,C 180,E1 -13532.33,E2 -13532.33} C_VEL
LIN {X 0,Y 354.797,Z 242.788,A -85,B 0,C 180,E1 -13535.696,E2 -13535.696} C_VEL
LIN {X 0,Y 354.832,Z 242.92,A -85,B 0,C 180,E1 -13539.591,E2 -13539.591} C_VEL
LIN {X 0,Y 356.988,Z 252.577,A -85,B 0,C 180,E1 -13542.373,E2 -13542.373} C_VEL
LIN {X 0,Y 358.339,Z 259.443,A -85,B 0,C 180,E1 -13544.178,E2 -13544.178} C_VEL
LIN {X 0,Y 360.104,Z 265.963,A -85,B 0,C 180,E1 -13544.481,E2 -13544.481} C_VEL
LIN {X 0,Y 364.48,Z 288.275,A -85,B 0,C 180,E1 -13545.279,E2 -13545.279} C_VEL
LIN {X 0,Y 362.816,Z 367.588,A -85,B 0,C 180,E1 -13546.914,E2 -13546.914} C_VEL
LIN {X 0,Y 362.16,Z 381.143,A -85,B 0,C 180,E1 -13547.426,E2 -13547.426} C_VEL
LIN {X 0,Y 361.355,Z 393.97,A -85,B 0,C 180,E1 -13548.154,E2 -13548.154} C_VEL
LIN {X 0,Y 360.426,Z 404.924,A -85,B 0,C 180,E1 -13548.989,E2 -13548.989} C_VEL
LIN {X 0,Y 359.201,Z 416.803,A -85,B 0,C 180,E1 -13550.152,E2 -13550.152} C_VEL
LIN {X 0,Y 358.1,Z 426.301,A -85,B 0,C 180,E1 -13551.316,E2 -13551.316} C_VEL
LIN {X 0,Y 356.947,Z 435.754,A -85,B 0,C 180,E1 -13552.741,E2 -13552.741} C_VEL
LIN {X 0,Y 355.904,Z 444.48,A -85,B 0,C 180,E1 -13554.384,E2 -13554.384} C_VEL
LIN {X 0,Y 354.922,Z 452.452,A -85,B 0,C 180,E1 -13556.26,E2 -13556.26} C_VEL
LIN {X 0,Y 354.189,Z 458.694,A -85,B 0,C 180,E1 -13558.156,E2 -13558.156} C_VEL
LIN {X 0,Y 353.663,Z 463.82,A -85,B 0,C 180,E1 -13560.213,E2 -13560.213} C_VEL
LIN {X 0,Y 353.408,Z 466.253,A -85,B 0,C 180,E1 -13561.494,E2 -13561.494} C_VEL
LIN {X 0,Y 353.112,Z 469,A -85,B 0,C 180,E1 -13563.577,E2 -13563.577} C_VEL
LIN {X 0,Y 352.963,Z 470.248,A -85,B 0,C 180,E1 -13565.284,E2 -13565.284} C_VEL
LIN {X 0,Y 352.941,Z 470.591,A -85,B 0,C 180,E1 -13566.532,E2 -13566.532} C_VEL
LIN {X 0,Y 352.91,Z 470.485,A -85,B 0,C 180,E1 -13567.768,E2 -13567.768} C_VEL
LIN {X 0,Y 352.982,Z 469.628,A -85,B 0,C 180,E1 -13569.34,E2 -13569.34} C_VEL
LIN {X 0,Y 353.201,Z 467.324,A -85,B 0,C 180,E1 -13571.437,E2 -13571.437} C_VEL
LIN {X 0,Y 353.467,Z 464.147,A -85,B 0,C 180,E1 -13573.253,E2 -13573.253} C_VEL
LIN {X 0,Y 353.841,Z 459.872,A -85,B 0,C 180,E1 -13575.037,E2 -13575.037} C_VEL
LIN {X 0,Y 354.419,Z 454.015,A -85,B 0,C 180,E1 -13576.907,E2 -13576.907} C_VEL
LIN {X 0,Y 355.091,Z 447.38,A -85,B 0,C 180,E1 -13578.586,E2 -13578.586} C_VEL
LIN {X 0,Y 356.063,Z 439.006,A -85,B 0,C 180,E1 -13580.286,E2 -13580.286} C_VEL
LIN {X 0,Y 357.059,Z 429.704,A -85,B 0,C 180,E1 -13581.797,E2 -13581.797} C_VEL
LIN {X 0,Y 358.122,Z 419.808,A -85,B 0,C 180,E1 -13583.097,E2 -13583.097} C_VEL
LIN {X 0,Y 359.185,Z 408.955,A -85,B 0,C 180,E1 -13584.246,E2 -13584.246} C_VEL
LIN {X 0,Y 360.176,Z 396.687,A -85,B 0,C 180,E1 -13585.253,E2 -13585.253} C_VEL
LIN {X 0,Y 360.933,Z 384.188,A -85,B 0,C 180,E1 -13586.023,E2 -13586.023} C_VEL
LIN {X 0,Y 361.593,Z 371.857,A -85,B 0,C 180,E1 -13586.554,E2 -13586.554} C_VEL
LIN {X 0,Y 361.996,Z 358.304,A -85,B 0,C 180,E1 -13586.904,E2 -13586.904} C_VEL
LIN {X 0,Y 363.156,Z 287.033,A -85,B 0,C 180,E1 -13588.342,E2 -13588.342} C_VEL
LIN {X 0,Y 357.981,Z 259.86,A -85,B 0,C 180,E1 -13589.249,E2 -13589.249} C_VEL
LIN {X 0,Y 357.879,Z 257.731,A -85,B 0,C 180,E1 -13589.72,E2 -13589.72} C_VEL
LIN {X 0,Y 356.34,Z 248.773,A -85,B 0,C 180,E1 -13592.262,E2 -13592.262} C_VEL
LIN {X 0,Y 354.919,Z 242.841,A -85,B 0,C 180,E1 -13594.082,E2 -13594.082} C_VEL
LIN {X 0,Y 355.091,Z 242.749,A -85,B 0,C 180,E1 -13596.821,E2 -13596.821} C_VEL
LIN {X 0,Y 354.953,Z 242.765,A -85,B 0,C 180,E1 -13599.365,E2 -13599.365} C_VEL
LIN {X 0,Y 354.261,Z 242.856,A -85,B 0,C 180,E1 -13600.311,E2 -13600.311} C_VEL
LIN {X 0,Y 351.415,Z 243.212,A -85,B 0,C 180,E1 -13601.851,E2 -13601.851} C_VEL
LIN {X 0,Y 349.004,Z 243.514,A -85,B 0,C 180,E1 -13603.096,E2 -13603.096} C_VEL
LIN {X 0,Y 347.947,Z 243.644,A -85,B 0,C 180,E1 -13604.06,E2 -13604.06} C_VEL
LIN {X 0,Y 347.848,Z 243.655,A -85,B 0,C 180,E1 -13604.386,E2 -13604.386} C_VEL
LIN {X 0,Y 347.859,Z 243.654,A -85,B 0,C 180,E1 -13608.292,E2 -13608.292} C_VEL
LIN {X 0,Y 347.733,Z 243.669,A -85,B 0,C 180,E1 -13611.627,E2 -13611.627} C_VEL
LIN {X 0,Y 347.742,Z 243.663,A -85,B 0,C 180,E1 -13615.115,E2 -13615.115} C_VEL
LIN {X 0,Y 347.711,Z 243.672,A -85,B 0,C 180,E1 -13617.703,E2 -13617.703} C_VEL
LIN {X 0,Y 347.707,Z 243.667,A -85,B 0,C 180,E1 -13620.353,E2 -13620.353} C_VEL
LIN {X 0,Y 347.722,Z 243.665,A -85,B 0,C 180,E1 -13624.047,E2 -13624.047} C_VEL
LIN {X 0,Y 347.729,Z 243.666,A -85,B 0,C 180,E1 -13627.326,E2 -13627.326} C_VEL
LIN {X 0,Y 347.672,Z 243.676,A -85,B 0,C 180,E1 -13630.306,E2 -13630.306} C_VEL
LIN {X 0,Y 347.698,Z 243.661,A -85,B 0,C 180,E1 -13633.413,E2 -13633.413} C_VEL
LIN {X 0,Y 347.702,Z 243.676,A -85,B 0,C 180,E1 -13636.691,E2 -13636.691} C_VEL
LIN {X 0,Y 347.682,Z 243.661,A -85,B 0,C 180,E1 -13640.187,E2 -13640.187} C_VEL
LIN {X 0,Y 347.738,Z 243.651,A -85,B 0,C 180,E1 -13642.683,E2 -13642.683} C_VEL
LIN {X 0,Y 347.733,Z 243.666,A -85,B 0,C 180,E1 -13645.961,E2 -13645.961} C_VEL
LIN {X 0,Y 347.723,Z 243.651,A -85,B 0,C 180,E1 -13649.655,E2 -13649.655} C_VEL
LIN {X 0,Y 347.725,Z 243.658,A -85,B 0,C 180,E1 -13653.604,E2 -13653.604} C_VEL
LIN {X 0,Y 347.742,Z 243.666,A -85,B 0,C 180,E1 -13656.164,E2 -13656.164} C_VEL
LIN {X 0,Y 347.799,Z 243.647,A -85,B 0,C 180,E1 -13659.913,E2 -13659.913} C_VEL
LIN {X 0,Y 347.827,Z 243.629,A -85,B 0,C 180,E1 -13663.573,E2 -13663.573} C_VEL
LIN {X 0,Y 347.884,Z 243.646,A -85,B 0,C 180,E1 -13667.165,E2 -13667.165} C_VEL
LIN {X 0,Y 347.932,Z 243.635,A -85,B 0,C 180,E1 -13670.705,E2 -13670.705} C_VEL
LIN {X 0,Y 348.036,Z 243.601,A -85,B 0,C 180,E1 -13674.209,E2 -13674.209} C_VEL
LIN {X 0,Y 348.19,Z 243.604,A -85,B 0,C 180,E1 -13677.69,E2 -13677.69} C_VEL
LIN {X 0,Y 348.14,Z 243.613,A -85,B 0,C 180,E1 -13681.161,E2 -13681.161} C_VEL
LIN {X 0,Y 348.184,Z 243.603,A -85,B 0,C 180,E1 -13682.317,E2 -13682.317} C_VEL
LIN {X 0,Y 348.077,Z 243.613,A -85,B 0,C 180,E1 -13686.962,E2 -13686.962} C_VEL
LIN {X 0,Y 347.901,Z 243.651,A -85,B 0,C 180,E1 -13690.479,E2 -13690.479} C_VEL
LIN {X 0,Y 347.907,Z 243.632,A -85,B 0,C 180,E1 -13694.153,E2 -13694.153} C_VEL
LIN {X 0,Y 347.838,Z 243.65,A -85,B 0,C 180,E1 -13698.262,E2 -13698.262} C_VEL
LIN {X 0,Y 347.777,Z 243.658,A -85,B 0,C 180,E1 -13701.629,E2 -13701.629} C_VEL
LIN {X 0,Y 347.779,Z 243.65,A -85,B 0,C 180,E1 -13705.114,E2 -13705.114} C_VEL
LIN {X 0,Y 347.747,Z 243.666,A -85,B 0,C 180,E1 -13707.703,E2 -13707.703} C_VEL
LIN {X 0,Y 347.75,Z 243.659,A -85,B 0,C 180,E1 -13710.351,E2 -13710.351} C_VEL
LIN {X 0,Y 347.761,Z 243.665,A -85,B 0,C 180,E1 -13714.046,E2 -13714.046} C_VEL
LIN {X 0,Y 347.768,Z 243.656,A -85,B 0,C 180,E1 -13717.323,E2 -13717.323} C_VEL
LIN {X 0,Y 347.753,Z 243.661,A -85,B 0,C 180,E1 -13721.602,E2 -13721.602} C_VEL
LIN {X 0,Y 347.714,Z 243.671,A -85,B 0,C 180,E1 -13725.029,E2 -13725.029} C_VEL
LIN {X 0,Y 347.754,Z 243.665,A -85,B 0,C 180,E1 -13728.4,E2 -13728.4} C_VEL
LIN {X 0,Y 347.769,Z 243.665,A -85,B 0,C 180,E1 -13732.679,E2 -13732.679} C_VEL
LIN {X 0,Y 347.762,Z 243.661,A -85,B 0,C 180,E1 -13735.957,E2 -13735.957} C_VEL
LIN {X 0,Y 347.763,Z 243.662,A -85,B 0,C 180,E1 -13739.653,E2 -13739.653} C_VEL
LIN {X 0,Y 347.814,Z 243.741,A -85,B 0,C 180,E1 -13740.539,E2 -13740.539} C_VEL
LIN {X 0,Y 349.639,Z 252.535,A -85,B 0,C 180,E1 -13743.11,E2 -13743.11} C_VEL
LIN {X 0,Y 351.434,Z 262.276,A -85,B 0,C 180,E1 -13745.797,E2 -13745.797} C_VEL
LIN {X 0,Y 350.913,Z 268.567,A -85,B 0,C 180,E1 -13747.323,E2 -13747.323} C_VEL
LIN {X 0,Y 352.156,Z 275.699,A -85,B 0,C 180,E1 -13747.604,E2 -13747.604} C_VEL
LIN {X 0,Y 356.408,Z 301.253,A -85,B 0,C 180,E1 -13748.413,E2 -13748.413} C_VEL
LIN {X 0,Y 354.989,Z 376.867,A -85,B 0,C 180,E1 -13749.992,E2 -13749.992} C_VEL
LIN {X 0,Y 354.334,Z 389.863,A -85,B 0,C 180,E1 -13750.482,E2 -13750.482} C_VEL
LIN {X 0,Y 353.502,Z 401.908,A -85,B 0,C 180,E1 -13751.151,E2 -13751.151} C_VEL
LIN {X 0,Y 352.514,Z 413.295,A -85,B 0,C 180,E1 -13751.999,E2 -13751.999} C_VEL
LIN {X 0,Y 351.362,Z 425.021,A -85,B 0,C 180,E1 -13753.139,E2 -13753.139} C_VEL
LIN {X 0,Y 350.321,Z 435.046,A -85,B 0,C 180,E1 -13754.363,E2 -13754.363} C_VEL
LIN {X 0,Y 349.35,Z 444.171,A -85,B 0,C 180,E1 -13755.732,E2 -13755.732} C_VEL
LIN {X 0,Y 348.419,Z 452.103,A -85,B 0,C 180,E1 -13757.18,E2 -13757.18} C_VEL
LIN {X 0,Y 347.546,Z 459.842,A -85,B 0,C 180,E1 -13758.923,E2 -13758.923} C_VEL
LIN {X 0,Y 346.941,Z 466.048,A -85,B 0,C 180,E1 -13760.673,E2 -13760.673} C_VEL
LIN {X 0,Y 346.492,Z 470.97,A -85,B 0,C 180,E1 -13762.423,E2 -13762.423} C_VEL
LIN {X 0,Y 346.261,Z 474.756,A -85,B 0,C 180,E1 -13764.174,E2 -13764.174} C_VEL
LIN {X 0,Y 346.173,Z 476.706,A -85,B 0,C 180,E1 -13765.341,E2 -13765.341} C_VEL
LIN {X 0,Y 346.129,Z 478.237,A -85,B 0,C 180,E1 -13766.507,E2 -13766.507} C_VEL
LIN {X 0,Y 346.054,Z 479.31,A -85,B 0,C 180,E1 -13767.671,E2 -13767.671} C_VEL
LIN {X 0,Y 346.056,Z 479.985,A -85,B 0,C 180,E1 -13768.835,E2 -13768.835} C_VEL
LIN {X 0,Y 346.082,Z 480.273,A -85,B 0,C 180,E1 -13769.999,E2 -13769.999} C_VEL
LIN {X 0,Y 346.056,Z 480.17,A -85,B 0,C 180,E1 -13771.163,E2 -13771.163} C_VEL
LIN {X 0,Y 346.134,Z 478.698,A -85,B 0,C 180,E1 -13773.491,E2 -13773.491} C_VEL
LIN {X 0,Y 346.197,Z 477.369,A -85,B 0,C 180,E1 -13774.657,E2 -13774.657} C_VEL
LIN {X 0,Y 346.29,Z 475.284,A -85,B 0,C 180,E1 -13776.014,E2 -13776.014} C_VEL
LIN {X 0,Y 346.661,Z 470.729,A -85,B 0,C 180,E1 -13778.158,E2 -13778.158} C_VEL
LIN {X 0,Y 347.157,Z 465.776,A -85,B 0,C 180,E1 -13779.908,E2 -13779.908} C_VEL
LIN {X 0,Y 347.886,Z 459.552,A -85,B 0,C 180,E1 -13781.654,E2 -13781.654} C_VEL
LIN {X 0,Y 348.954,Z 451.793,A -85,B 0,C 180,E1 -13783.391,E2 -13783.391} C_VEL
LIN {X 0,Y 349.998,Z 443.869,A -85,B 0,C 180,E1 -13784.833,E2 -13784.833} C_VEL
LIN {X 0,Y 351.088,Z 434.212,A -85,B 0,C 180,E1 -13786.274,E2 -13786.274} C_VEL
LIN {X 0,Y 352.231,Z 424.79,A -85,B 0,C 180,E1 -13787.414,E2 -13787.414} C_VEL
LIN {X 0,Y 353.517,Z 413.127,A -85,B 0,C 180,E1 -13788.546,E2 -13788.546} C_VEL
LIN {X 0,Y 354.66,Z 400.692,A -85,B 0,C 180,E1 -13789.459,E2 -13789.459} C_VEL
LIN {X 0,Y 355.624,Z 387.63,A -85,B 0,C 180,E1 -13790.157,E2 -13790.157} C_VEL
LIN {X 0,Y 356.265,Z 374.695,A -85,B 0,C 180,E1 -13790.609,E2 -13790.609} C_VEL
LIN {X 0,Y 357.703,Z 301.197,A -85,B 0,C 180,E1 -13792.147,E2 -13792.147} C_VEL
LIN {X 0,Y 353.87,Z 279.592,A -85,B 0,C 180,E1 -13792.909,E2 -13792.909} C_VEL
LIN {X 0,Y 351.598,Z 268.372,A -85,B 0,C 180,E1 -13793.363,E2 -13793.363} C_VEL
LIN {X 0,Y 351.768,Z 265.977,A -85,B 0,C 180,E1 -13793.863,E2 -13793.863} C_VEL
LIN {X 0,Y 351.689,Z 262.316,A -85,B 0,C 180,E1 -13794.812,E2 -13794.812} C_VEL
LIN {X 0,Y 349.623,Z 251.559,A -85,B 0,C 180,E1 -13797.809,E2 -13797.809} C_VEL
LIN {X 0,Y 347.835,Z 243.771,A -85,B 0,C 180,E1 -13800.145,E2 -13800.145} C_VEL
LIN {X 0,Y 347.751,Z 243.666,A -85,B 0,C 180,E1 -13804.462,E2 -13804.462} C_VEL
LIN {X 0,Y 347.768,Z 243.665,A -85,B 0,C 180,E1 -13807.984,E2 -13807.984} C_VEL
LIN {X 0,Y 347.749,Z 243.667,A -85,B 0,C 180,E1 -13811.829,E2 -13811.829} C_VEL
LIN {X 0,Y 347.709,Z 243.671,A -85,B 0,C 180,E1 -13815.024,E2 -13815.024} C_VEL
LIN {X 0,Y 347.745,Z 243.666,A -85,B 0,C 180,E1 -13818.396,E2 -13818.396} C_VEL
LIN {X 0,Y 347.758,Z 243.668,A -85,B 0,C 180,E1 -13822.675,E2 -13822.675} C_VEL
LIN {X 0,Y 347.75,Z 243.664,A -85,B 0,C 180,E1 -13825.953,E2 -13825.953} C_VEL
LIN {X 0,Y 347.739,Z 243.665,A -85,B 0,C 180,E1 -13829.648,E2 -13829.648} C_VEL
LIN {X 0,Y 347.739,Z 243.665,A -85,B 0,C 180,E1 -13833.597,E2 -13833.597} C_VEL
LIN {X 0,Y 347.765,Z 243.662,A -85,B 0,C 180,E1 -13836.157,E2 -13836.157} C_VEL
LIN {X 0,Y 347.804,Z 243.658,A -85,B 0,C 180,E1 -13839.905,E2 -13839.905} C_VEL
LIN {X 0,Y 347.829,Z 243.658,A -85,B 0,C 180,E1 -13843.565,E2 -13843.565} C_VEL
LIN {X 0,Y 347.885,Z 243.643,A -85,B 0,C 180,E1 -13847.157,E2 -13847.157} C_VEL
LIN {X 0,Y 347.929,Z 243.641,A -85,B 0,C 180,E1 -13850.697,E2 -13850.697} C_VEL
LIN {X 0,Y 348.062,Z 243.625,A -85,B 0,C 180,E1 -13853.038,E2 -13853.038} C_VEL
LIN {X 0,Y 348.171,Z 243.612,A -85,B 0,C 180,E1 -13857.682,E2 -13857.682} C_VEL
LIN {X 0,Y 348.105,Z 243.615,A -85,B 0,C 180,E1 -13861.153,E2 -13861.153} C_VEL
LIN {X 0,Y 348.145,Z 243.616,A -85,B 0,C 180,E1 -13862.31,E2 -13862.31} C_VEL
LIN {X 0,Y 348.037,Z 243.628,A -85,B 0,C 180,E1 -13866.955,E2 -13866.955} C_VEL
LIN {X 0,Y 347.877,Z 243.65,A -85,B 0,C 180,E1 -13870.472,E2 -13870.472} C_VEL
LIN {X 0,Y 347.884,Z 243.649,A -85,B 0,C 180,E1 -13874.146,E2 -13874.146} C_VEL
LIN {X 0,Y 347.813,Z 243.662,A -85,B 0,C 180,E1 -13878.255,E2 -13878.255} C_VEL
LIN {X 0,Y 347.749,Z 243.668,A -85,B 0,C 180,E1 -13881.622,E2 -13881.622} C_VEL
LIN {X 0,Y 347.753,Z 243.664,A -85,B 0,C 180,E1 -13885.108,E2 -13885.108} C_VEL
LIN {X 0,Y 347.718,Z 243.668,A -85,B 0,C 180,E1 -13887.696,E2 -13887.696} C_VEL
LIN {X 0,Y 347.716,Z 243.673,A -85,B 0,C 180,E1 -13890.345,E2 -13890.345} C_VEL
LIN {X 0,Y 347.724,Z 243.673,A -85,B 0,C 180,E1 -13894.04,E2 -13894.04} C_VEL
LIN {X 0,Y 347.738,Z 243.666,A -85,B 0,C 180,E1 -13897.317,E2 -13897.317} C_VEL
LIN {X 0,Y 347.762,Z 243.737,A -85,B 0,C 180,E1 -13899.097,E2 -13899.097} C_VEL
LIN {X 0,Y 349.328,Z 250.67,A -85,B 0,C 180,E1 -13901.208,E2 -13901.208} C_VEL
LIN {X 0,Y 351.169,Z 259.483,A -85,B 0,C 180,E1 -13903.633,E2 -13903.633} C_VEL
LIN {X 0,Y 353.35,Z 265.941,A -85,B 0,C 180,E1 -13903.985,E2 -13903.985} C_VEL
LIN {X 0,Y 357.879,Z 288.834,A -85,B 0,C 180,E1 -13904.832,E2 -13904.832} C_VEL
LIN {X 0,Y 356.244,Z 367.079,A -85,B 0,C 180,E1 -13906.476,E2 -13906.476} C_VEL
LIN {X 0,Y 355.568,Z 380.689,A -85,B 0,C 180,E1 -13906.99,E2 -13906.99} C_VEL
LIN {X 0,Y 354.703,Z 393.943,A -85,B 0,C 180,E1 -13907.747,E2 -13907.747} C_VEL
LIN {X 0,Y 353.678,Z 405.487,A -85,B 0,C 180,E1 -13908.647,E2 -13908.647} C_VEL
LIN {X 0,Y 352.463,Z 416.948,A -85,B 0,C 180,E1 -13909.795,E2 -13909.795} C_VEL
LIN {X 0,Y 351.14,Z 427.707,A -85,B 0,C 180,E1 -13911.155,E2 -13911.155} C_VEL
LIN {X 0,Y 349.961,Z 436.803,A -85,B 0,C 180,E1 -13912.594,E2 -13912.594} C_VEL
LIN {X 0,Y 348.886,Z 445.315,A -85,B 0,C 180,E1 -13914.257,E2 -13914.257} C_VEL
LIN {X 0,Y 348.017,Z 452.052,A -85,B 0,C 180,E1 -13915.881,E2 -13915.881} C_VEL
LIN {X 0,Y 347.298,Z 457.716,A -85,B 0,C 180,E1 -13917.572,E2 -13917.572} C_VEL
LIN {X 0,Y 346.742,Z 462.881,A -85,B 0,C 180,E1 -13919.556,E2 -13919.556} C_VEL
LIN {X 0,Y 346.319,Z 466.605,A -85,B 0,C 180,E1 -13921.519,E2 -13921.519} C_VEL
LIN {X 0,Y 346.047,Z 469.082,A -85,B 0,C 180,E1 -13923.462,E2 -13923.462} C_VEL
LIN {X 0,Y 345.882,Z 470.103,A -85,B 0,C 180,E1 -13924.743,E2 -13924.743} C_VEL
LIN {X 0,Y 345.82,Z 470.642,A -85,B 0,C 180,E1 -13926.124,E2 -13926.124} C_VEL
LIN {X 0,Y 345.811,Z 470.66,A -85,B 0,C 180,E1 -13927.287,E2 -13927.287} C_VEL
LIN {X 0,Y 345.887,Z 469.867,A -85,B 0,C 180,E1 -13929.157,E2 -13929.157} C_VEL
LIN {X 0,Y 346.062,Z 468.017,A -85,B 0,C 180,E1 -13931.04,E2 -13931.04} C_VEL
LIN {X 0,Y 346.246,Z 465.782,A -85,B 0,C 180,E1 -13932.533,E2 -13932.533} C_VEL
LIN {X 0,Y 346.674,Z 461.137,A -85,B 0,C 180,E1 -13934.721,E2 -13934.721} C_VEL
LIN {X 0,Y 347.285,Z 455.29,A -85,B 0,C 180,E1 -13936.741,E2 -13936.741} C_VEL
LIN {X 0,Y 348.024,Z 448.099,A -85,B 0,C 180,E1 -13938.646,E2 -13938.646} C_VEL
LIN {X 0,Y 348.973,Z 440.172,A -85,B 0,C 180,E1 -13940.321,E2 -13940.321} C_VEL
LIN {X 0,Y 350.051,Z 430.762,A -85,B 0,C 180,E1 -13941.922,E2 -13941.922} C_VEL
LIN {X 0,Y 351.264,Z 419.848,A -85,B 0,C 180,E1 -13943.395,E2 -13943.395} C_VEL
LIN {X 0,Y 352.326,Z 409.496,A -85,B 0,C 180,E1 -13944.513,E2 -13944.513} C_VEL
LIN {X 0,Y 353.263,Z 398.773,A -85,B 0,C 180,E1 -13945.437,E2 -13945.437} C_VEL
LIN {X 0,Y 354.015,Z 386.784,A -85,B 0,C 180,E1 -13946.23,E2 -13946.23} C_VEL
LIN {X 0,Y 354.775,Z 373.615,A -85,B 0,C 180,E1 -13946.843,E2 -13946.843} C_VEL
LIN {X 0,Y 355.207,Z 361.37,A -85,B 0,C 180,E1 -13947.201,E2 -13947.201} C_VEL
LIN {X 0,Y 356.494,Z 288.023,A -85,B 0,C 180,E1 -13948.711,E2 -13948.711} C_VEL
LIN {X 0,Y 351.271,Z 260.891,A -85,B 0,C 180,E1 -13949.627,E2 -13949.627} C_VEL
LIN {X 0,Y 350.971,Z 259.424,A -85,B 0,C 180,E1 -13949.743,E2 -13949.743} C_VEL
LIN {X 0,Y 349.449,Z 250.463,A -85,B 0,C 180,E1 -13952.306,E2 -13952.306} C_VEL
LIN {X 0,Y 347.853,Z 243.7,A -85,B 0,C 180,E1 -13954.419,E2 -13954.419} C_VEL
LIN {X 0,Y 348.057,Z 243.626,A -85,B 0,C 180,E1 -13956.96,E2 -13956.96} C_VEL
LIN {X 0,Y 347.897,Z 243.649,A -85,B 0,C 180,E1 -13960.476,E2 -13960.476} C_VEL
LIN {X 0,Y 347.848,Z 243.655,A -85,B 0,C 180,E1 -13964.386,E2 -13964.386} C_VEL
LIN {X 0,Y 347.154,Z 243.743,A -85,B 0,C 180,E1 -13965.352,E2 -13965.352} C_VEL
LIN {X 0,Y 344.314,Z 244.095,A -85,B 0,C 180,E1 -13966.924,E2 -13966.924} C_VEL
LIN {X 0,Y 341.904,Z 244.396,A -85,B 0,C 180,E1 -13968.196,E2 -13968.196} C_VEL
LIN {X 0,Y 340.838,Z 244.527,A -85,B 0,C 180,E1 -13969.18,E2 -13969.18} C_VEL
LIN {X 0,Y 340.732,Z 244.538,A -85,B 0,C 180,E1 -13969.514,E2 -13969.514} C_VEL
LIN {X 0,Y 340.679,Z 244.545,A -85,B 0,C 180,E1 -13973.077,E2 -13973.077} C_VEL
LIN {X 0,Y 340.694,Z 244.543,A -85,B 0,C 180,E1 -13975.672,E2 -13975.672} C_VEL
LIN {X 0,Y 340.674,Z 244.536,A -85,B 0,C 180,E1 -13979.678,E2 -13979.678} C_VEL
LIN {X 0,Y 340.658,Z 244.552,A -85,B 0,C 180,E1 -13982.44,E2 -13982.44} C_VEL
LIN {X 0,Y 340.689,Z 244.53,A -85,B 0,C 180,E1 -13985.283,E2 -13985.283} C_VEL
LIN {X 0,Y 340.669,Z 244.551,A -85,B 0,C 180,E1 -13988.386,E2 -13988.386} C_VEL
LIN {X 0,Y 340.667,Z 244.535,A -85,B 0,C 180,E1 -13992.048,E2 -13992.048} C_VEL
LIN {X 0,Y 340.629,Z 244.552,A -85,B 0,C 180,E1 -13996.232,E2 -13996.232} C_VEL
LIN {X 0,Y 340.649,Z 244.547,A -85,B 0,C 180,E1 -13998.692,E2 -13998.692} C_VEL
LIN {X 0,Y 340.701,Z 244.523,A -85,B 0,C 180,E1 -14001.775,E2 -14001.775} C_VEL
LIN {X 0,Y 340.707,Z 244.543,A -85,B 0,C 180,E1 -14005.6,E2 -14005.6} C_VEL
LIN {X 0,Y 340.679,Z 244.536,A -85,B 0,C 180,E1 -14008.959,E2 -14008.959} C_VEL
LIN {X 0,Y 340.699,Z 244.525,A -85,B 0,C 180,E1 -14013.017,E2 -14013.017} C_VEL
LIN {X 0,Y 340.696,Z 244.545,A -85,B 0,C 180,E1 -14016.93,E2 -14016.93} C_VEL
LIN {X 0,Y 340.756,Z 244.521,A -85,B 0,C 180,E1 -14020.736,E2 -14020.736} C_VEL
LIN {X 0,Y 340.813,Z 244.516,A -85,B 0,C 180,E1 -14024.455,E2 -14024.455} C_VEL
LIN {X 0,Y 340.843,Z 244.527,A -85,B 0,C 180,E1 -14028.105,E2 -14028.105} C_VEL
LIN {X 0,Y 340.979,Z 244.495,A -85,B 0,C 180,E1 -14031.709,E2 -14031.709} C_VEL
LIN {X 0,Y 341.012,Z 244.475,A -85,B 0,C 180,E1 -14034.09,E2 -14034.09} C_VEL
LIN {X 0,Y 341.127,Z 244.483,A -85,B 0,C 180,E1 -14037.643,E2 -14037.643} C_VEL
LIN {X 0,Y 341.109,Z 244.488,A -85,B 0,C 180,E1 -14041.185,E2 -14041.185} C_VEL
LIN {X 0,Y 341.121,Z 244.482,A -85,B 0,C 180,E1 -14042.365,E2 -14042.365} C_VEL
LIN {X 0,Y 341.046,Z 244.49,A -85,B 0,C 180,E1 -14047.106,E2 -14047.106} C_VEL
LIN {X 0,Y 340.853,Z 244.528,A -85,B 0,C 180,E1 -14050.698,E2 -14050.698} C_VEL
LIN {X 0,Y 340.872,Z 244.506,A -85,B 0,C 180,E1 -14054.328,E2 -14054.328} C_VEL
LIN {X 0,Y 340.795,Z 244.529,A -85,B 0,C 180,E1 -14058.443,E2 -14058.443} C_VEL
LIN {X 0,Y 340.728,Z 244.535,A -85,B 0,C 180,E1 -14061.844,E2 -14061.844} C_VEL
LIN {X 0,Y 340.73,Z 244.536,A -85,B 0,C 180,E1 -14065.671,E2 -14065.671} C_VEL
LIN {X 0,Y 340.716,Z 244.536,A -85,B 0,C 180,E1 -14069.677,E2 -14069.677} C_VEL
LIN {X 0,Y 340.698,Z 244.536,A -85,B 0,C 180,E1 -14072.438,E2 -14072.438} C_VEL
LIN {X 0,Y 340.729,Z 244.543,A -85,B 0,C 180,E1 -14075.281,E2 -14075.281} C_VEL
LIN {X 0,Y 340.706,Z 244.538,A -85,B 0,C 180,E1 -14078.384,E2 -14078.384} C_VEL
LIN {X 0,Y 340.706,Z 244.535,A -85,B 0,C 180,E1 -14082.046,E2 -14082.046} C_VEL
LIN {X 0,Y 340.663,Z 244.545,A -85,B 0,C 180,E1 -14086.229,E2 -14086.229} C_VEL
LIN {X 0,Y 340.683,Z 244.545,A -85,B 0,C 180,E1 -14088.689,E2 -14088.689} C_VEL
LIN {X 0,Y 340.732,Z 244.541,A -85,B 0,C 180,E1 -14091.772,E2 -14091.772} C_VEL
LIN {X 0,Y 340.737,Z 244.54,A -85,B 0,C 180,E1 -14095.596,E2 -14095.596} C_VEL
LIN {X 0,Y 340.711,Z 244.541,A -85,B 0,C 180,E1 -14098.956,E2 -14098.956} C_VEL
LIN {X 0,Y 340.774,Z 244.696,A -85,B 0,C 180,E1 -14100.241,E2 -14100.241} C_VEL
LIN {X 0,Y 342.644,Z 253.603,A -85,B 0,C 180,E1 -14102.872,E2 -14102.872} C_VEL
LIN {X 0,Y 344.451,Z 263.256,A -85,B 0,C 180,E1 -14105.595,E2 -14105.595} C_VEL
LIN {X 0,Y 344.091,Z 268.454,A -85,B 0,C 180,E1 -14106.883,E2 -14106.883} C_VEL
LIN {X 0,Y 345.493,Z 276.624,A -85,B 0,C 180,E1 -14107.205,E2 -14107.205} C_VEL
LIN {X 0,Y 349.729,Z 302.506,A -85,B 0,C 180,E1 -14108.042,E2 -14108.042} C_VEL
LIN {X 0,Y 348.248,Z 376.85,A -85,B 0,C 180,E1 -14109.627,E2 -14109.627} C_VEL
LIN {X 0,Y 347.586,Z 389.818,A -85,B 0,C 180,E1 -14110.126,E2 -14110.126} C_VEL
LIN {X 0,Y 346.684,Z 402.413,A -85,B 0,C 180,E1 -14110.842,E2 -14110.842} C_VEL
LIN {X 0,Y 345.576,Z 414.422,A -85,B 0,C 180,E1 -14111.778,E2 -14111.778} C_VEL
LIN {X 0,Y 344.39,Z 425.918,A -85,B 0,C 180,E1 -14112.94,E2 -14112.94} C_VEL
LIN {X 0,Y 343.361,Z 435.584,A -85,B 0,C 180,E1 -14114.164,E2 -14114.164} C_VEL
LIN {X 0,Y 342.218,Z 445.583,A -85,B 0,C 180,E1 -14115.732,E2 -14115.732} C_VEL
LIN {X 0,Y 341.114,Z 454.603,A -85,B 0,C 180,E1 -14117.505,E2 -14117.505} C_VEL
LIN {X 0,Y 340.316,Z 461.865,A -85,B 0,C 180,E1 -14119.288,E2 -14119.288} C_VEL
LIN {X 0,Y 339.73,Z 467.656,A -85,B 0,C 180,E1 -14121.073,E2 -14121.073} C_VEL
LIN {X 0,Y 339.333,Z 472.207,A -85,B 0,C 180,E1 -14122.861,E2 -14122.861} C_VEL
LIN {X 0,Y 339.182,Z 474.6,A -85,B 0,C 180,E1 -14124.052,E2 -14124.052} C_VEL
LIN {X 0,Y 339.079,Z 476.56,A -85,B 0,C 180,E1 -14125.243,E2 -14125.243} C_VEL
LIN {X 0,Y 339.056,Z 478.104,A -85,B 0,C 180,E1 -14126.434,E2 -14126.434} C_VEL
LIN {X 0,Y 338.97,Z 479.191,A -85,B 0,C 180,E1 -14127.622,E2 -14127.622} C_VEL
LIN {X 0,Y 338.962,Z 479.874,A -85,B 0,C 180,E1 -14128.811,E2 -14128.811} C_VEL
LIN {X 0,Y 338.985,Z 480.17,A -85,B 0,C 180,E1 -14129.999,E2 -14129.999} C_VEL
LIN {X 0,Y 338.962,Z 480.078,A -85,B 0,C 180,E1 -14131.187,E2 -14131.187} C_VEL
LIN {X 0,Y 338.971,Z 479.555,A -85,B 0,C 180,E1 -14132.376,E2 -14132.376} C_VEL
LIN {X 0,Y 339.062,Z 478.629,A -85,B 0,C 180,E1 -14133.564,E2 -14133.564} C_VEL
LIN {X 0,Y 339.101,Z 477.308,A -85,B 0,C 180,E1 -14134.754,E2 -14134.754} C_VEL
LIN {X 0,Y 339.261,Z 474.516,A -85,B 0,C 180,E1 -14136.541,E2 -14136.541} C_VEL
LIN {X 0,Y 339.61,Z 470.702,A -85,B 0,C 180,E1 -14138.328,E2 -14138.328} C_VEL
LIN {X 0,Y 340.14,Z 465.767,A -85,B 0,C 180,E1 -14140.114,E2 -14140.114} C_VEL
LIN {X 0,Y 340.901,Z 459.564,A -85,B 0,C 180,E1 -14141.896,E2 -14141.896} C_VEL
LIN {X 0,Y 342.028,Z 451.841,A -85,B 0,C 180,E1 -14143.667,E2 -14143.667} C_VEL
LIN {X 0,Y 343.118,Z 443.945,A -85,B 0,C 180,E1 -14145.137,E2 -14145.137} C_VEL
LIN {X 0,Y 344.274,Z 434.322,A -85,B 0,C 180,E1 -14146.605,E2 -14146.605} C_VEL
LIN {X 0,Y 345.664,Z 423.654,A -85,B 0,C 180,E1 -14147.909,E2 -14147.909} C_VEL
LIN {X 0,Y 346.806,Z 413.36,A -85,B 0,C 180,E1 -14148.918,E2 -14148.918} C_VEL
LIN {X 0,Y 347.996,Z 401.075,A -85,B 0,C 180,E1 -14149.848,E2 -14149.848} C_VEL
LIN {X 0,Y 349.038,Z 387.447,A -85,B 0,C 180,E1 -14150.593,E2 -14150.593} C_VEL
LIN {X 0,Y 349.703,Z 374.47,A -85,B 0,C 180,E1 -14151.052,E2 -14151.052} C_VEL
LIN {X 0,Y 351.25,Z 302.271,A -85,B 0,C 180,E1 -14152.589,E2 -14152.589} C_VEL
LIN {X 0,Y 346.947,Z 278.197,A -85,B 0,C 180,E1 -14153.466,E2 -14153.466} C_VEL
LIN {X 0,Y 344.874,Z 268.069,A -85,B 0,C 180,E1 -14153.913,E2 -14153.913} C_VEL
LIN {X 0,Y 344.966,Z 264.822,A -85,B 0,C 180,E1 -14154.685,E2 -14154.685} C_VEL
LIN {X 0,Y 343.17,Z 255.081,A -85,B 0,C 180,E1 -14157.437,E2 -14157.437} C_VEL
LIN {X 0,Y 340.746,Z 244.664,A -85,B 0,C 180,E1 -14160.611,E2 -14160.611} C_VEL
LIN {X 0,Y 340.73,Z 244.539,A -85,B 0,C 180,E1 -14164.402,E2 -14164.402} C_VEL
LIN {X 0,Y 340.725,Z 244.546,A -85,B 0,C 180,E1 -14168.227,E2 -14168.227} C_VEL
LIN {X 0,Y 340.699,Z 244.547,A -85,B 0,C 180,E1 -14172.042,E2 -14172.042} C_VEL
LIN {X 0,Y 340.656,Z 244.55,A -85,B 0,C 180,E1 -14176.224,E2 -14176.224} C_VEL
LIN {X 0,Y 340.675,Z 244.547,A -85,B 0,C 180,E1 -14178.685,E2 -14178.685} C_VEL
LIN {X 0,Y 340.721,Z 244.536,A -85,B 0,C 180,E1 -14181.768,E2 -14181.768} C_VEL
LIN {X 0,Y 340.724,Z 244.539,A -85,B 0,C 180,E1 -14185.593,E2 -14185.593} C_VEL
LIN {X 0,Y 340.694,Z 244.542,A -85,B 0,C 180,E1 -14188.952,E2 -14188.952} C_VEL
LIN {X 0,Y 340.712,Z 244.538,A -85,B 0,C 180,E1 -14193.009,E2 -14193.009} C_VEL
LIN {X 0,Y 340.74,Z 244.537,A -85,B 0,C 180,E1 -14195.634,E2 -14195.634} C_VEL
LIN {X 0,Y 340.733,Z 244.541,A -85,B 0,C 180,E1 -14199.47,E2 -14199.47} C_VEL
LIN {X 0,Y 340.791,Z 244.524,A -85,B 0,C 180,E1 -14201.977,E2 -14201.977} C_VEL
LIN {X 0,Y 340.85,Z 244.519,A -85,B 0,C 180,E1 -14205.713,E2 -14205.713} C_VEL
LIN {X 0,Y 340.841,Z 244.53,A -85,B 0,C 180,E1 -14209.302,E2 -14209.302} C_VEL
LIN {X 0,Y 341.007,Z 244.502,A -85,B 0,C 180,E1 -14212.893,E2 -14212.893} C_VEL
LIN {X 0,Y 340.803,Z 244.529,A -85,B 0,C 180,E1 -14215.265,E2 -14215.265} C_VEL
LIN {X 0,Y 341.108,Z 244.491,A -85,B 0,C 180,E1 -14217.634,E2 -14217.634} C_VEL
LIN {X 0,Y 341.076,Z 244.49,A -85,B 0,C 180,E1 -14221.177,E2 -14221.177} C_VEL
LIN {X 0,Y 341.085,Z 244.495,A -85,B 0,C 180,E1 -14222.358,E2 -14222.358} C_VEL
LIN {X 0,Y 340.973,Z 244.505,A -85,B 0,C 180,E1 -14226.467,E2 -14226.467} C_VEL
LIN {X 0,Y 340.867,Z 244.52,A -85,B 0,C 180,E1 -14229.49,E2 -14229.49} C_VEL
LIN {X 0,Y 340.828,Z 244.526,A -85,B 0,C 180,E1 -14233.106,E2 -14233.106} C_VEL
LIN {X 0,Y 340.801,Z 244.535,A -85,B 0,C 180,E1 -14235.546,E2 -14235.546} C_VEL
LIN {X 0,Y 340.745,Z 244.54,A -85,B 0,C 180,E1 -14239.264,E2 -14239.264} C_VEL
LIN {X 0,Y 340.695,Z 244.543,A -85,B 0,C 180,E1 -14243.07,E2 -14243.07} C_VEL
LIN {X 0,Y 340.704,Z 244.542,A -85,B 0,C 180,E1 -14245.664,E2 -14245.664} C_VEL
LIN {X 0,Y 340.683,Z 244.544,A -85,B 0,C 180,E1 -14249.671,E2 -14249.671} C_VEL
LIN {X 0,Y 340.663,Z 244.544,A -85,B 0,C 180,E1 -14252.432,E2 -14252.432} C_VEL
LIN {X 0,Y 340.694,Z 244.542,A -85,B 0,C 180,E1 -14255.275,E2 -14255.275} C_VEL
LIN {X 0,Y 340.706,Z 244.65,A -85,B 0,C 180,E1 -14258.647,E2 -14258.647} C_VEL
LIN {X 0,Y 342.764,Z 253.547,A -85,B 0,C 180,E1 -14261.388,E2 -14261.388} C_VEL
LIN {X 0,Y 343.977,Z 259.548,A -85,B 0,C 180,E1 -14263.056,E2 -14263.056} C_VEL
LIN {X 0,Y 346.943,Z 267.317,A -85,B 0,C 180,E1 -14263.523,E2 -14263.523} C_VEL
LIN {X 0,Y 351.401,Z 289.808,A -85,B 0,C 180,E1 -14264.38,E2 -14264.38} C_VEL
LIN {X 0,Y 349.713,Z 366.941,A -85,B 0,C 180,E1 -14266.03,E2 -14266.03} C_VEL
LIN {X 0,Y 348.991,Z 380.594,A -85,B 0,C 180,E1 -14266.55,E2 -14266.55} C_VEL
LIN {X 0,Y 348.184,Z 392.944,A -85,B 0,C 180,E1 -14267.259,E2 -14267.259} C_VEL
LIN {X 0,Y 347.22,Z 403.853,A -85,B 0,C 180,E1 -14268.093,E2 -14268.093} C_VEL
LIN {X 0,Y 346.044,Z 414.733,A -85,B 0,C 180,E1 -14269.158,E2 -14269.158} C_VEL
LIN {X 0,Y 344.711,Z 425.074,A -85,B 0,C 180,E1 -14270.424,E2 -14270.424} C_VEL
LIN {X 0,Y 343.384,Z 435.011,A -85,B 0,C 180,E1 -14271.936,E2 -14271.936} C_VEL
LIN {X 0,Y 342.294,Z 443.098,A -85,B 0,C 180,E1 -14273.458,E2 -14273.458} C_VEL
LIN {X 0,Y 341.269,Z 450.584,A -85,B 0,C 180,E1 -14275.202,E2 -14275.202} C_VEL
LIN {X 0,Y 340.34,Z 457.311,A -85,B 0,C 180,E1 -14277.177,E2 -14277.177} C_VEL
LIN {X 0,Y 339.806,Z 461.818,A -85,B 0,C 180,E1 -14278.866,E2 -14278.866} C_VEL
LIN {X 0,Y 339.463,Z 465.043,A -85,B 0,C 180,E1 -14280.393,E2 -14280.393} C_VEL
LIN {X 0,Y 339.213,Z 466.961,A -85,B 0,C 180,E1 -14281.543,E2 -14281.543} C_VEL
LIN {X 0,Y 338.983,Z 468.895,A -85,B 0,C 180,E1 -14283.05,E2 -14283.05} C_VEL
LIN {X 0,Y 338.835,Z 469.879,A -85,B 0,C 180,E1 -14284.179,E2 -14284.179} C_VEL
LIN {X 0,Y 338.723,Z 470.718,A -85,B 0,C 180,E1 -14285.9,E2 -14285.9} C_VEL
LIN {X 0,Y 338.708,Z 470.551,A -85,B 0,C 180,E1 -14288.07,E2 -14288.07} C_VEL
LIN {X 0,Y 338.813,Z 469.841,A -85,B 0,C 180,E1 -14289.353,E2 -14289.353} C_VEL
LIN {X 0,Y 338.897,Z 468.69,A -85,B 0,C 180,E1 -14290.623,E2 -14290.623} C_VEL
LIN {X 0,Y 339.16,Z 466.28,A -85,B 0,C 180,E1 -14292.383,E2 -14292.383} C_VEL
LIN {X 0,Y 339.5,Z 462.337,A -85,B 0,C 180,E1 -14294.39,E2 -14294.39} C_VEL
LIN {X 0,Y 340.022,Z 457.42,A -85,B 0,C 180,E1 -14296.252,E2 -14296.252} C_VEL
LIN {X 0,Y 340.697,Z 451.194,A -85,B 0,C 180,E1 -14298.096,E2 -14298.096} C_VEL
LIN {X 0,Y 341.678,Z 443.128,A -85,B 0,C 180,E1 -14299.992,E2 -14299.992} C_VEL
LIN {X 0,Y 342.602,Z 435.434,A -85,B 0,C 180,E1 -14301.448,E2 -14301.448} C_VEL
LIN {X 0,Y 343.725,Z 425.648,A -85,B 0,C 180,E1 -14302.954,E2 -14302.954} C_VEL
LIN {X 0,Y 344.901,Z 414.815,A -85,B 0,C 180,E1 -14304.293,E2 -14304.293} C_VEL
LIN {X 0,Y 346.005,Z 404.145,A -85,B 0,C 180,E1 -14305.341,E2 -14305.341} C_VEL
LIN {X 0,Y 346.928,Z 392.597,A -85,B 0,C 180,E1 -14306.226,E2 -14306.226} C_VEL
LIN {X 0,Y 347.674,Z 380.359,A -85,B 0,C 180,E1 -14306.923,E2 -14306.923} C_VEL
LIN {X 0,Y 348.354,Z 366.875,A -85,B 0,C 180,E1 -14307.435,E2 -14307.435} C_VEL
LIN {X 0,Y 349.763,Z 288.291,A -85,B 0,C 180,E1 -14309.111,E2 -14309.111} C_VEL
LIN {X 0,Y 344.643,Z 262.165,A -85,B 0,C 180,E1 -14310.015,E2 -14310.015} C_VEL
LIN {X 0,Y 343.898,Z 259.561,A -85,B 0,C 180,E1 -14310.187,E2 -14310.187} C_VEL
LIN {X 0,Y 342.156,Z 250.194,A -85,B 0,C 180,E1 -14312.944,E2 -14312.944} C_VEL
LIN {X 0,Y 340.839,Z 244.604,A -85,B 0,C 180,E1 -14314.732,E2 -14314.732} C_VEL
LIN {X 0,Y 341.025,Z 244.502,A -85,B 0,C 180,E1 -14317.104,E2 -14317.104} C_VEL
LIN {X 0,Y 340.839,Z 244.528,A -85,B 0,C 180,E1 -14320.696,E2 -14320.696} C_VEL
LIN {X 0,Y 340.827,Z 244.53,A -85,B 0,C 180,E1 -14324.368,E2 -14324.368} C_VEL
LIN {X 0,Y 340.805,Z 244.531,A -85,B 0,C 180,E1 -14328.469,E2 -14328.469} C_VEL
LIN {X 0,Y 340.732,Z 244.538,A -85,B 0,C 180,E1 -14329.514,E2 -14329.514} C_VEL
LIN {X 0,Y 340.001,Z 244.63,A -85,B 0,C 180,E1 -14330.499,E2 -14330.499} C_VEL
LIN {X 0,Y 337.091,Z 244.997,A -85,B 0,C 180,E1 -14332.102,E2 -14332.102} C_VEL
LIN {X 0,Y 334.691,Z 245.291,A -85,B 0,C 180,E1 -14333.4,E2 -14333.4} C_VEL
LIN {X 0,Y 333.709,Z 245.41,A -85,B 0,C 180,E1 -14334.405,E2 -14334.405} C_VEL
LIN {X 0,Y 333.653,Z 245.417,A -85,B 0,C 180,E1 -14334.745,E2 -14334.745} C_VEL
LIN {X 0,Y 333.626,Z 245.426,A -85,B 0,C 180,E1 -14337.792,E2 -14337.792} C_VEL
LIN {X 0,Y 333.628,Z 245.42,A -85,B 0,C 180,E1 -14340.37,E2 -14340.37} C_VEL
LIN {X 0,Y 333.61,Z 245.425,A -85,B 0,C 180,E1 -14343.212,E2 -14343.212} C_VEL
LIN {X 0,Y 333.647,Z 245.411,A -85,B 0,C 180,E1 -14346.143,E2 -14346.143} C_VEL
LIN {X 0,Y 333.577,Z 245.431,A -85,B 0,C 180,E1 -14349.203,E2 -14349.203} C_VEL
LIN {X 0,Y 333.603,Z 245.412,A -85,B 0,C 180,E1 -14352.503,E2 -14352.503} C_VEL
LIN {X 0,Y 333.573,Z 245.43,A -85,B 0,C 180,E1 -14355.959,E2 -14355.959} C_VEL
LIN {X 0,Y 333.583,Z 245.419,A -85,B 0,C 180,E1 -14359.329,E2 -14359.329} C_VEL
LIN {X 0,Y 333.645,Z 245.411,A -85,B 0,C 180,E1 -14363.173,E2 -14363.173} C_VEL
LIN {X 0,Y 333.657,Z 245.423,A -85,B 0,C 180,E1 -14365.346,E2 -14365.346} C_VEL
LIN {X 0,Y 333.615,Z 245.42,A -85,B 0,C 180,E1 -14368.226,E2 -14368.226} C_VEL
LIN {X 0,Y 333.616,Z 245.4,A -85,B 0,C 180,E1 -14371.025,E2 -14371.025} C_VEL
LIN {X 0,Y 333.649,Z 245.417,A -85,B 0,C 180,E1 -14374.926,E2 -14374.926} C_VEL
LIN {X 0,Y 333.659,Z 245.418,A -85,B 0,C 180,E1 -14379.023,E2 -14379.023} C_VEL
LIN {X 0,Y 333.736,Z 245.382,A -85,B 0,C 180,E1 -14381.591,E2 -14381.591} C_VEL
LIN {X 0,Y 333.805,Z 245.393,A -85,B 0,C 180,E1 -14385.581,E2 -14385.581} C_VEL
LIN {X 0,Y 333.812,Z 245.4,A -85,B 0,C 180,E1 -14389.082,E2 -14389.082} C_VEL
LIN {X 0,Y 333.954,Z 245.36,A -85,B 0,C 180,E1 -14392.75,E2 -14392.75} C_VEL
LIN {X 0,Y 333.777,Z 245.38,A -85,B 0,C 180,E1 -14395.173,E2 -14395.173} C_VEL
LIN {X 0,Y 334.067,Z 245.362,A -85,B 0,C 180,E1 -14397.593,E2 -14397.593} C_VEL
LIN {X 0,Y 334.078,Z 245.364,A -85,B 0,C 180,E1 -14401.209,E2 -14401.209} C_VEL
LIN {X 0,Y 334.061,Z 245.36,A -85,B 0,C 180,E1 -14402.416,E2 -14402.416} C_VEL
LIN {X 0,Y 334.005,Z 245.351,A -85,B 0,C 180,E1 -14406.043,E2 -14406.043} C_VEL
LIN {X 0,Y 333.826,Z 245.399,A -85,B 0,C 180,E1 -14409.7,E2 -14409.7} C_VEL
LIN {X 0,Y 333.8,Z 245.392,A -85,B 0,C 180,E1 -14413.395,E2 -14413.395} C_VEL
LIN {X 0,Y 333.728,Z 245.403,A -85,B 0,C 180,E1 -14417.151,E2 -14417.151} C_VEL
LIN {X 0,Y 333.695,Z 245.416,A -85,B 0,C 180,E1 -14419.697,E2 -14419.697} C_VEL
LIN {X 0,Y 333.669,Z 245.399,A -85,B 0,C 180,E1 -14423.594,E2 -14423.594} C_VEL
LIN {X 0,Y 333.667,Z 245.415,A -85,B 0,C 180,E1 -14426.256,E2 -14426.256} C_VEL
LIN {X 0,Y 333.673,Z 245.412,A -85,B 0,C 180,E1 -14430.28,E2 -14430.28} C_VEL
LIN {X 0,Y 333.649,Z 245.42,A -85,B 0,C 180,E1 -14433.211,E2 -14433.211} C_VEL
LIN {X 0,Y 333.687,Z 245.413,A -85,B 0,C 180,E1 -14436.141,E2 -14436.141} C_VEL
LIN {X 0,Y 333.614,Z 245.425,A -85,B 0,C 180,E1 -14439.201,E2 -14439.201} C_VEL
LIN {X 0,Y 333.641,Z 245.414,A -85,B 0,C 180,E1 -14442.501,E2 -14442.501} C_VEL
LIN {X 0,Y 333.607,Z 245.425,A -85,B 0,C 180,E1 -14445.956,E2 -14445.956} C_VEL
LIN {X 0,Y 333.615,Z 245.426,A -85,B 0,C 180,E1 -14449.326,E2 -14449.326} C_VEL
LIN {X 0,Y 333.676,Z 245.421,A -85,B 0,C 180,E1 -14453.17,E2 -14453.17} C_VEL
LIN {X 0,Y 333.687,Z 245.421,A -85,B 0,C 180,E1 -14455.342,E2 -14455.342} C_VEL
LIN {X 0,Y 333.705,Z 245.412,A -85,B 0,C 180,E1 -14459.638,E2 -14459.638} C_VEL
LIN {X 0,Y 333.806,Z 245.993,A -85,B 0,C 180,E1 -14460.034,E2 -14460.034} C_VEL
LIN {X 0,Y 335.857,Z 255.684,A -85,B 0,C 180,E1 -14462.926,E2 -14462.926} C_VEL
LIN {X 0,Y 337.452,Z 264.238,A -85,B 0,C 180,E1 -14465.383,E2 -14465.383} C_VEL
LIN {X 0,Y 337.255,Z 268.406,A -85,B 0,C 180,E1 -14466.43,E2 -14466.43} C_VEL
LIN {X 0,Y 340.547,Z 286.958,A -85,B 0,C 180,E1 -14467.116,E2 -14467.116} C_VEL
LIN {X 0,Y 343.033,Z 302.297,A -85,B 0,C 180,E1 -14467.624,E2 -14467.624} C_VEL
LIN {X 0,Y 341.568,Z 375.687,A -85,B 0,C 180,E1 -14469.21,E2 -14469.21} C_VEL
LIN {X 0,Y 340.902,Z 389.014,A -85,B 0,C 180,E1 -14469.719,E2 -14469.719} C_VEL
LIN {X 0,Y 339.965,Z 401.789,A -85,B 0,C 180,E1 -14470.449,E2 -14470.449} C_VEL
LIN {X 0,Y 338.829,Z 413.955,A -85,B 0,C 180,E1 -14471.402,E2 -14471.402} C_VEL
LIN {X 0,Y 337.595,Z 425.519,A -85,B 0,C 180,E1 -14472.586,E2 -14472.586} C_VEL
LIN {X 0,Y 336.407,Z 436.109,A -85,B 0,C 180,E1 -14473.954,E2 -14473.954} C_VEL
LIN {X 0,Y 335.291,Z 445.295,A -85,B 0,C 180,E1 -14475.431,E2 -14475.431} C_VEL
LIN {X 0,Y 334.168,Z 454.35,A -85,B 0,C 180,E1 -14477.241,E2 -14477.241} C_VEL
LIN {X 0,Y 333.317,Z 461.639,A -85,B 0,C 180,E1 -14479.06,E2 -14479.06} C_VEL
LIN {X 0,Y 332.678,Z 467.462,A -85,B 0,C 180,E1 -14480.883,E2 -14480.883} C_VEL
LIN {X 0,Y 332.272,Z 472.036,A -85,B 0,C 180,E1 -14482.708,E2 -14482.708} C_VEL
LIN {X 0,Y 332.077,Z 474.782,A -85,B 0,C 180,E1 -14484.118,E2 -14484.118} C_VEL
LIN {X 0,Y 331.961,Z 477.967,A -85,B 0,C 180,E1 -14486.358,E2 -14486.358} C_VEL
LIN {X 0,Y 331.89,Z 479.071,A -85,B 0,C 180,E1 -14487.572,E2 -14487.572} C_VEL
LIN {X 0,Y 331.871,Z 479.763,A -85,B 0,C 180,E1 -14488.786,E2 -14488.786} C_VEL
LIN {X 0,Y 331.891,Z 480.067,A -85,B 0,C 180,E1 -14489.999,E2 -14489.999} C_VEL
LIN {X 0,Y 331.87,Z 479.984,A -85,B 0,C 180,E1 -14491.212,E2 -14491.212} C_VEL
LIN {X 0,Y 331.89,Z 479.478,A -85,B 0,C 180,E1 -14492.426,E2 -14492.426} C_VEL
LIN {X 0,Y 331.969,Z 478.56,A -85,B 0,C 180,E1 -14493.64,E2 -14493.64} C_VEL
LIN {X 0,Y 332.079,Z 475.807,A -85,B 0,C 180,E1 -14495.887,E2 -14495.887} C_VEL
LIN {X 0,Y 332.416,Z 472.08,A -85,B 0,C 180,E1 -14497.898,E2 -14497.898} C_VEL
LIN {X 0,Y 332.925,Z 467.553,A -85,B 0,C 180,E1 -14499.722,E2 -14499.722} C_VEL
LIN {X 0,Y 333.808,Z 460.698,A -85,B 0,C 180,E1 -14501.845,E2 -14501.845} C_VEL
LIN {X 0,Y 334.932,Z 453.274,A -85,B 0,C 180,E1 -14503.653,E2 -14503.653} C_VEL
LIN {X 0,Y 336.248,Z 444.046,A -85,B 0,C 180,E1 -14505.454,E2 -14505.454} C_VEL
LIN {X 0,Y 337.459,Z 434.475,A -85,B 0,C 180,E1 -14506.951,E2 -14506.951} C_VEL
LIN {X 0,Y 338.928,Z 423.868,A -85,B 0,C 180,E1 -14508.277,E2 -14508.277} C_VEL
LIN {X 0,Y 340.316,Z 411.981,A -85,B 0,C 180,E1 -14509.45,E2 -14509.45} C_VEL
LIN {X 0,Y 341.446,Z 400.398,A -85,B 0,C 180,E1 -14510.323,E2 -14510.323} C_VEL
LIN {X 0,Y 342.498,Z 387.327,A -85,B 0,C 180,E1 -14511.044,E2 -14511.044} C_VEL
LIN {X 0,Y 343.167,Z 374.343,A -85,B 0,C 180,E1 -14511.512,E2 -14511.512} C_VEL
LIN {X 0,Y 344.791,Z 303.213,A -85,B 0,C 180,E1 -14513.053,E2 -14513.053} C_VEL
LIN {X 0,Y 340.713,Z 280.153,A -85,B 0,C 180,E1 -14513.919,E2 -14513.919} C_VEL
LIN {X 0,Y 338.193,Z 268.32,A -85,B 0,C 180,E1 -14514.437,E2 -14514.437} C_VEL
LIN {X 0,Y 338.159,Z 267.403,A -85,B 0,C 180,E1 -14514.56,E2 -14514.56} C_VEL
LIN {X 0,Y 336.471,Z 257.587,A -85,B 0,C 180,E1 -14517.355,E2 -14517.355} C_VEL
LIN {X 0,Y 334.183,Z 247.531,A -85,B 0,C 180,E1 -14520.426,E2 -14520.426} C_VEL
LIN {X 0,Y 333.675,Z 245.447,A -85,B 0,C 180,E1 -14521.196,E2 -14521.196} C_VEL
LIN {X 0,Y 333.692,Z 245.419,A -85,B 0,C 180,E1 -14524.771,E2 -14524.771} C_VEL
LIN {X 0,Y 333.649,Z 245.421,A -85,B 0,C 180,E1 -14527.65,E2 -14527.65} C_VEL
LIN {X 0,Y 333.609,Z 245.421,A -85,B 0,C 180,E1 -14530.771,E2 -14530.771} C_VEL
LIN {X 0,Y 333.597,Z 245.432,A -85,B 0,C 180,E1 -14534.247,E2 -14534.247} C_VEL
LIN {X 0,Y 333.642,Z 245.425,A -85,B 0,C 180,E1 -14537.615,E2 -14537.615} C_VEL
LIN {X 0,Y 333.619,Z 245.421,A -85,B 0,C 180,E1 -14541.207,E2 -14541.207} C_VEL
LIN {X 0,Y 333.676,Z 245.42,A -85,B 0,C 180,E1 -14543.857,E2 -14543.857} C_VEL
LIN {X 0,Y 333.646,Z 245.422,A -85,B 0,C 180,E1 -14547.41,E2 -14547.41} C_VEL
LIN {X 0,Y 333.652,Z 245.423,A -85,B 0,C 180,E1 -14551.019,E2 -14551.019} C_VEL
LIN {X 0,Y 333.694,Z 245.419,A -85,B 0,C 180,E1 -14555.085,E2 -14555.085} C_VEL
LIN {X 0,Y 333.666,Z 245.423,A -85,B 0,C 180,E1 -14559.015,E2 -14559.015} C_VEL
LIN {X 0,Y 333.74,Z 245.402,A -85,B 0,C 180,E1 -14561.583,E2 -14561.583} C_VEL
LIN {X 0,Y 333.806,Z 245.397,A -85,B 0,C 180,E1 -14565.573,E2 -14565.573} C_VEL
LIN {X 0,Y 333.811,Z 245.405,A -85,B 0,C 180,E1 -14569.074,E2 -14569.074} C_VEL
LIN {X 0,Y 333.96,Z 245.379,A -85,B 0,C 180,E1 -14572.742,E2 -14572.742} C_VEL
LIN {X 0,Y 333.771,Z 245.406,A -85,B 0,C 180,E1 -14575.165,E2 -14575.165} C_VEL
LIN {X 0,Y 334.048,Z 245.369,A -85,B 0,C 180,E1 -14577.584,E2 -14577.584} C_VEL
LIN {X 0,Y 334.046,Z 245.365,A -85,B 0,C 180,E1 -14581.201,E2 -14581.201} C_VEL
LIN {X 0,Y 333.774,Z 245.411,A -85,B 0,C 180,E1 -14583.617,E2 -14583.617} C_VEL
LIN {X 0,Y 333.944,Z 245.381,A -85,B 0,C 180,E1 -14586.458,E2 -14586.458} C_VEL
LIN {X 0,Y 333.805,Z 245.399,A -85,B 0,C 180,E1 -14589.692,E2 -14589.692} C_VEL
LIN {X 0,Y 333.781,Z 245.403,A -85,B 0,C 180,E1 -14593.387,E2 -14593.387} C_VEL
LIN {X 0,Y 333.702,Z 245.411,A -85,B 0,C 180,E1 -14597.144,E2 -14597.144} C_VEL
LIN {X 0,Y 333.7,Z 245.417,A -85,B 0,C 180,E1 -14599.688,E2 -14599.688} C_VEL
LIN {X 0,Y 333.641,Z 245.422,A -85,B 0,C 180,E1 -14603.587,E2 -14603.587} C_VEL
LIN {X 0,Y 333.64,Z 245.426,A -85,B 0,C 180,E1 -14606.249,E2 -14606.249} C_VEL
LIN {X 0,Y 333.639,Z 245.426,A -85,B 0,C 180,E1 -14610.274,E2 -14610.274} C_VEL
LIN {X 0,Y 333.613,Z 245.427,A -85,B 0,C 180,E1 -14613.205,E2 -14613.205} C_VEL
LIN {X 0,Y 333.652,Z 245.425,A -85,B 0,C 180,E1 -14616.135,E2 -14616.135} C_VEL
LIN {X 0,Y 333.683,Z 245.509,A -85,B 0,C 180,E1 -14618.141,E2 -14618.141} C_VEL
LIN {X 0,Y 335.651,Z 254.142,A -85,B 0,C 180,E1 -14620.875,E2 -14620.875} C_VEL
LIN {X 0,Y 336.841,Z 259.743,A -85,B 0,C 180,E1 -14622.471,E2 -14622.471} C_VEL
LIN {X 0,Y 340.946,Z 270.314,A -85,B 0,C 180,E1 -14623.107,E2 -14623.107} C_VEL
LIN {X 0,Y 345.035,Z 291.225,A -85,B 0,C 180,E1 -14623.929,E2 -14623.929} C_VEL
LIN {X 0,Y 343.159,Z 367.515,A -85,B 0,C 180,E1 -14625.587,E2 -14625.587} C_VEL
LIN {X 0,Y 342.409,Z 381.25,A -85,B 0,C 180,E1 -14626.129,E2 -14626.129} C_VEL
LIN {X 0,Y 341.569,Z 393.226,A -85,B 0,C 180,E1 -14626.834,E2 -14626.834} C_VEL
LIN {X 0,Y 340.418,Z 405.386,A -85,B 0,C 180,E1 -14627.802,E2 -14627.802} C_VEL
LIN {X 0,Y 339.022,Z 417.301,A -85,B 0,C 180,E1 -14629.037,E2 -14629.037} C_VEL
LIN {X 0,Y 337.633,Z 427.447,A -85,B 0,C 180,E1 -14630.361,E2 -14630.361} C_VEL
LIN {X 0,Y 336.273,Z 437.071,A -85,B 0,C 180,E1 -14631.938,E2 -14631.938} C_VEL
LIN {X 0,Y 335.112,Z 445.573,A -85,B 0,C 180,E1 -14633.67,E2 -14633.67} C_VEL
LIN {X 0,Y 334.087,Z 452.42,A -85,B 0,C 180,E1 -14635.392,E2 -14635.392} C_VEL
LIN {X 0,Y 333.27,Z 458.198,A -85,B 0,C 180,E1 -14637.203,E2 -14637.203} C_VEL
LIN {X 0,Y 332.728,Z 462.33,A -85,B 0,C 180,E1 -14638.837,E2 -14638.837} C_VEL
LIN {X 0,Y 332.264,Z 466.312,A -85,B 0,C 180,E1 -14640.891,E2 -14640.891} C_VEL
LIN {X 0,Y 331.92,Z 468.831,A -85,B 0,C 180,E1 -14642.772,E2 -14642.772} C_VEL
LIN {X 0,Y 331.692,Z 470.487,A -85,B 0,C 180,E1 -14644.929,E2 -14644.929} C_VEL
LIN {X 0,Y 331.61,Z 470.869,A -85,B 0,C 180,E1 -14646.256,E2 -14646.256} C_VEL
LIN {X 0,Y 331.591,Z 470.811,A -85,B 0,C 180,E1 -14647.574,E2 -14647.574} C_VEL
LIN {X 0,Y 331.666,Z 470.261,A -85,B 0,C 180,E1 -14648.887,E2 -14648.887} C_VEL
LIN {X 0,Y 331.752,Z 469.25,A -85,B 0,C 180,E1 -14650.188,E2 -14650.188} C_VEL
LIN {X 0,Y 332.047,Z 466.707,A -85,B 0,C 180,E1 -14652.242,E2 -14652.242} C_VEL
LIN {X 0,Y 332.337,Z 463.438,A -85,B 0,C 180,E1 -14654.044,E2 -14654.044} C_VEL
LIN {X 0,Y 332.903,Z 458.238,A -85,B 0,C 180,E1 -14656.171,E2 -14656.171} C_VEL
LIN {X 0,Y 333.618,Z 451.84,A -85,B 0,C 180,E1 -14658.149,E2 -14658.149} C_VEL
LIN {X 0,Y 334.57,Z 444.174,A -85,B 0,C 180,E1 -14660.021,E2 -14660.021} C_VEL
LIN {X 0,Y 335.583,Z 436.327,A -85,B 0,C 180,E1 -14661.571,E2 -14661.571} C_VEL
LIN {X 0,Y 336.749,Z 426.767,A -85,B 0,C 180,E1 -14663.109,E2 -14663.109} C_VEL
LIN {X 0,Y 337.961,Z 416.074,A -85,B 0,C 180,E1 -14664.482,E2 -14664.482} C_VEL
LIN {X 0,Y 339.209,Z 404.143,A -85,B 0,C 180,E1 -14665.694,E2 -14665.694} C_VEL
LIN {X 0,Y 340.19,Z 392.534,A -85,B 0,C 180,E1 -14666.596,E2 -14666.596} C_VEL
LIN {X 0,Y 340.973,Z 380.231,A -85,B 0,C 180,E1 -14667.306,E2 -14667.306} C_VEL
LIN {X 0,Y 341.582,Z 367.878,A -85,B 0,C 180,E1 -14667.79,E2 -14667.79} C_VEL
LIN {X 0,Y 343.224,Z 290.441,A -85,B 0,C 180,E1 -14669.471,E2 -14669.471} C_VEL
LIN {X 0,Y 338.477,Z 265.197,A -85,B 0,C 180,E1 -14670.353,E2 -14670.353} C_VEL
LIN {X 0,Y 336.798,Z 259.8,A -85,B 0,C 180,E1 -14670.637,E2 -14670.637} C_VEL
LIN {X 0,Y 335.269,Z 251.879,A -85,B 0,C 180,E1 -14673.005,E2 -14673.005} C_VEL
LIN {X 0,Y 333.844,Z 245.452,A -85,B 0,C 180,E1 -14675.096,E2 -14675.096} C_VEL
LIN {X 0,Y 333.972,Z 245.382,A -85,B 0,C 180,E1 -14677.255,E2 -14677.255} C_VEL
LIN {X 0,Y 333.802,Z 245.405,A -85,B 0,C 180,E1 -14680.924,E2 -14680.924} C_VEL
LIN {X 0,Y 333.776,Z 245.407,A -85,B 0,C 180,E1 -14684.637,E2 -14684.637} C_VEL
LIN {X 0,Y 333.764,Z 245.407,A -85,B 0,C 180,E1 -14688.657,E2 -14688.657} C_VEL
LIN {X 0,Y 333.622,Z 245.427,A -85,B 0,C 180,E1 -14692.284,E2 -14692.284} C_VEL
LIN {X 0,Y 333.653,Z 245.417,A -85,B 0,C 180,E1 -14694.745,E2 -14694.745} C_VEL
LIN {X 0,Y 333.038,Z 245.5,A -85,B 0,C 180,E1 -14695.753,E2 -14695.753} C_VEL
LIN {X 0,Y 330.159,Z 245.857,A -85,B 0,C 180,E1 -14697.391,E2 -14697.391} C_VEL
LIN {X 0,Y 327.689,Z 246.155,A -85,B 0,C 180,E1 -14698.719,E2 -14698.719} C_VEL
LIN {X 0,Y 326.638,Z 246.284,A -85,B 0,C 180,E1 -14699.748,E2 -14699.748} C_VEL
LIN {X 0,Y 326.56,Z 246.297,A -85,B 0,C 180,E1 -14700.097,E2 -14700.097} C_VEL
LIN {X 0,Y 326.58,Z 246.297,A -85,B 0,C 180,E1 -14704.024,E2 -14704.024} C_VEL
LIN {X 0,Y 326.597,Z 246.299,A -85,B 0,C 180,E1 -14707.241,E2 -14707.241} C_VEL
LIN {X 0,Y 326.52,Z 246.3,A -85,B 0,C 180,E1 -14711.128,E2 -14711.128} C_VEL
LIN {X 0,Y 326.537,Z 246.296,A -85,B 0,C 180,E1 -14713.531,E2 -14713.531} C_VEL
LIN {X 0,Y 326.551,Z 246.308,A -85,B 0,C 180,E1 -14717.034,E2 -14717.034} C_VEL
LIN {X 0,Y 326.553,Z 246.285,A -85,B 0,C 180,E1 -14720.786,E2 -14720.786} C_VEL
LIN {X 0,Y 326.595,Z 246.296,A -85,B 0,C 180,E1 -14724.485,E2 -14724.485} C_VEL
LIN {X 0,Y 326.594,Z 246.298,A -85,B 0,C 180,E1 -14727.46,E2 -14727.46} C_VEL
LIN {X 0,Y 326.567,Z 246.282,A -85,B 0,C 180,E1 -14730.338,E2 -14730.338} C_VEL
LIN {X 0,Y 326.585,Z 246.284,A -85,B 0,C 180,E1 -14733.139,E2 -14733.139} C_VEL
LIN {X 0,Y 326.602,Z 246.301,A -85,B 0,C 180,E1 -14735.873,E2 -14735.873} C_VEL
LIN {X 0,Y 326.625,Z 246.283,A -85,B 0,C 180,E1 -14739.868,E2 -14739.868} C_VEL
LIN {X 0,Y 326.658,Z 246.257,A -85,B 0,C 180,E1 -14742.475,E2 -14742.475} C_VEL
LIN {X 0,Y 326.753,Z 246.278,A -85,B 0,C 180,E1 -14746.319,E2 -14746.319} C_VEL
LIN {X 0,Y 326.78,Z 246.273,A -85,B 0,C 180,E1 -14750.097,E2 -14750.097} C_VEL
LIN {X 0,Y 326.94,Z 246.226,A -85,B 0,C 180,E1 -14753.834,E2 -14753.834} C_VEL
LIN {X 0,Y 327.01,Z 246.241,A -85,B 0,C 180,E1 -14757.541,E2 -14757.541} C_VEL
LIN {X 0,Y 327.046,Z 246.24,A -85,B 0,C 180,E1 -14761.235,E2 -14761.235} C_VEL
LIN {X 0,Y 326.742,Z 246.264,A -85,B 0,C 180,E1 -14763.704,E2 -14763.704} C_VEL
LIN {X 0,Y 326.961,Z 246.229,A -85,B 0,C 180,E1 -14766.174,E2 -14766.174} C_VEL
LIN {X 0,Y 326.789,Z 246.276,A -85,B 0,C 180,E1 -14769.911,E2 -14769.911} C_VEL
LIN {X 0,Y 326.764,Z 246.268,A -85,B 0,C 180,E1 -14773.689,E2 -14773.689} C_VEL
LIN {X 0,Y 326.673,Z 246.285,A -85,B 0,C 180,E1 -14777.533,E2 -14777.533} C_VEL
LIN {X 0,Y 326.641,Z 246.296,A -85,B 0,C 180,E1 -14780.14,E2 -14780.14} C_VEL
LIN {X 0,Y 326.642,Z 246.273,A -85,B 0,C 180,E1 -14784.133,E2 -14784.133} C_VEL
LIN {X 0,Y 326.613,Z 246.298,A -85,B 0,C 180,E1 -14788.086,E2 -14788.086} C_VEL
LIN {X 0,Y 326.584,Z 246.29,A -85,B 0,C 180,E1 -14791.1,E2 -14791.1} C_VEL
LIN {X 0,Y 326.619,Z 246.299,A -85,B 0,C 180,E1 -14794.022,E2 -14794.022} C_VEL
LIN {X 0,Y 326.635,Z 246.288,A -85,B 0,C 180,E1 -14797.239,E2 -14797.239} C_VEL
LIN {X 0,Y 326.557,Z 246.308,A -85,B 0,C 180,E1 -14801.126,E2 -14801.126} C_VEL
LIN {X 0,Y 326.573,Z 246.3,A -85,B 0,C 180,E1 -14803.528,E2 -14803.528} C_VEL
LIN {X 0,Y 326.586,Z 246.299,A -85,B 0,C 180,E1 -14807.03,E2 -14807.03} C_VEL
LIN {X 0,Y 326.585,Z 246.304,A -85,B 0,C 180,E1 -14810.783,E2 -14810.783} C_VEL
LIN {X 0,Y 326.625,Z 246.3,A -85,B 0,C 180,E1 -14814.481,E2 -14814.481} C_VEL
LIN {X 0,Y 326.622,Z 246.296,A -85,B 0,C 180,E1 -14817.456,E2 -14817.456} C_VEL
LIN {X 0,Y 326.692,Z 246.489,A -85,B 0,C 180,E1 -14819.511,E2 -14819.511} C_VEL
LIN {X 0,Y 329.074,Z 257.838,A -85,B 0,C 180,E1 -14823.009,E2 -14823.009} C_VEL
LIN {X 0,Y 330.591,Z 266.396,A -85,B 0,C 180,E1 -14825.509,E2 -14825.509} C_VEL
LIN {X 0,Y 330.45,Z 268.323,A -85,B 0,C 180,E1 -14825.959,E2 -14825.959} C_VEL
LIN {X 0,Y 332.863,Z 281.831,A -85,B 0,C 180,E1 -14826.486,E2 -14826.486} C_VEL
LIN {X 0,Y 336.438,Z 303.903,A -85,B 0,C 180,E1 -14827.238,E2 -14827.238} C_VEL
LIN {X 0,Y 334.84,Z 376.734,A -85,B 0,C 180,E1 -14828.853,E2 -14828.853} C_VEL
LIN {X 0,Y 334.144,Z 389.675,A -85,B 0,C 180,E1 -14829.371,E2 -14829.371} C_VEL
LIN {X 0,Y 333.172,Z 402.256,A -85,B 0,C 180,E1 -14830.113,E2 -14830.113} C_VEL
LIN {X 0,Y 332.086,Z 413.466,A -85,B 0,C 180,E1 -14831.01,E2 -14831.01} C_VEL
LIN {X 0,Y 330.81,Z 425.106,A -85,B 0,C 180,E1 -14832.217,E2 -14832.217} C_VEL
LIN {X 0,Y 329.61,Z 435.267,A -85,B 0,C 180,E1 -14833.541,E2 -14833.541} C_VEL
LIN {X 0,Y 328.389,Z 445.007,A -85,B 0,C 180,E1 -14835.118,E2 -14835.118} C_VEL
LIN {X 0,Y 327.231,Z 454.096,A -85,B 0,C 180,E1 -14836.966,E2 -14836.966} C_VEL
LIN {X 0,Y 326.296,Z 461.413,A -85,B 0,C 180,E1 -14838.822,E2 -14838.822} C_VEL
LIN {X 0,Y 325.643,Z 467.266,A -85,B 0,C 180,E1 -14840.684,E2 -14840.684} C_VEL
LIN {X 0,Y 325.206,Z 471.864,A -85,B 0,C 180,E1 -14842.549,E2 -14842.549} C_VEL
LIN {X 0,Y 324.989,Z 474.913,A -85,B 0,C 180,E1 -14844.157,E2 -14844.157} C_VEL
LIN {X 0,Y 324.87,Z 477.828,A -85,B 0,C 180,E1 -14846.278,E2 -14846.278} C_VEL
LIN {X 0,Y 324.812,Z 478.951,A -85,B 0,C 180,E1 -14847.519,E2 -14847.519} C_VEL
LIN {X 0,Y 324.783,Z 479.651,A -85,B 0,C 180,E1 -14848.759,E2 -14848.759} C_VEL
LIN {X 0,Y 324.8,Z 479.964,A -85,B 0,C 180,E1 -14849.999,E2 -14849.999} C_VEL
LIN {X 0,Y 324.782,Z 479.89,A -85,B 0,C 180,E1 -14851.239,E2 -14851.239} C_VEL
LIN {X 0,Y 324.812,Z 479.4,A -85,B 0,C 180,E1 -14852.479,E2 -14852.479} C_VEL
LIN {X 0,Y 324.878,Z 478.49,A -85,B 0,C 180,E1 -14853.72,E2 -14853.72} C_VEL
LIN {X 0,Y 325.052,Z 475.48,A -85,B 0,C 180,E1 -14856.205,E2 -14856.205} C_VEL
LIN {X 0,Y 325.367,Z 472.051,A -85,B 0,C 180,E1 -14858.07,E2 -14858.07} C_VEL
LIN {X 0,Y 325.9,Z 467.549,A -85,B 0,C 180,E1 -14859.933,E2 -14859.933} C_VEL
LIN {X 0,Y 326.84,Z 460.737,A -85,B 0,C 180,E1 -14862.101,E2 -14862.101} C_VEL
LIN {X 0,Y 328.025,Z 453.341,A -85,B 0,C 180,E1 -14863.946,E2 -14863.946} C_VEL
LIN {X 0,Y 329.393,Z 444.163,A -85,B 0,C 180,E1 -14865.784,E2 -14865.784} C_VEL
LIN {X 0,Y 330.674,Z 434.636,A -85,B 0,C 180,E1 -14867.309,E2 -14867.309} C_VEL
LIN {X 0,Y 332.18,Z 424.082,A -85,B 0,C 180,E1 -14868.662,E2 -14868.662} C_VEL
LIN {X 0,Y 333.654,Z 412.307,A -85,B 0,C 180,E1 -14869.854,E2 -14869.854} C_VEL
LIN {X 0,Y 334.935,Z 399.721,A -85,B 0,C 180,E1 -14870.817,E2 -14870.817} C_VEL
LIN {X 0,Y 336.004,Z 386.446,A -85,B 0,C 180,E1 -14871.551,E2 -14871.551} C_VEL
LIN {X 0,Y 336.732,Z 372.747,A -85,B 0,C 180,E1 -14872.025,E2 -14872.025} C_VEL
LIN {X 0,Y 338.361,Z 304.26,A -85,B 0,C 180,E1 -14873.533,E2 -14873.533} C_VEL
LIN {X 0,Y 334.113,Z 280.31,A -85,B 0,C 180,E1 -14874.469,E2 -14874.469} C_VEL
LIN {X 0,Y 331.49,Z 268.869,A -85,B 0,C 180,E1 -14874.988,E2 -14874.988} C_VEL
LIN {X 0,Y 331.152,Z 267.579,A -85,B 0,C 180,E1 -14875.115,E2 -14875.115} C_VEL
LIN {X 0,Y 329.302,Z 257.692,A -85,B 0,C 180,E1 -14878.002,E2 -14878.002} C_VEL
LIN {X 0,Y 326.708,Z 246.859,A -85,B 0,C 180,E1 -14881.442,E2 -14881.442} C_VEL
LIN {X 0,Y 326.62,Z 246.304,A -85,B 0,C 180,E1 -14881.813,E2 -14881.813} C_VEL
LIN {X 0,Y 326.619,Z 246.301,A -85,B 0,C 180,E1 -14885.517,E2 -14885.517} C_VEL
LIN {X 0,Y 326.594,Z 246.297,A -85,B 0,C 180,E1 -14889.219,E2 -14889.219} C_VEL
LIN {X 0,Y 326.579,Z 246.301,A -85,B 0,C 180,E1 -14892.968,E2 -14892.968} C_VEL
LIN {X 0,Y 326.578,Z 246.305,A -85,B 0,C 180,E1 -14897.026,E2 -14897.026} C_VEL
LIN {X 0,Y 326.575,Z 246.301,A -85,B 0,C 180,E1 -14900.778,E2 -14900.778} C_VEL
LIN {X 0,Y 326.613,Z 246.296,A -85,B 0,C 180,E1 -14904.477,E2 -14904.477} C_VEL
LIN {X 0,Y 326.61,Z 246.298,A -85,B 0,C 180,E1 -14907.452,E2 -14907.452} C_VEL
LIN {X 0,Y 326.616,Z 246.299,A -85,B 0,C 180,E1 -14910.333,E2 -14910.333} C_VEL
LIN {X 0,Y 326.641,Z 246.297,A -85,B 0,C 180,E1 -14914.641,E2 -14914.641} C_VEL
LIN {X 0,Y 326.615,Z 246.296,A -85,B 0,C 180,E1 -14918.539,E2 -14918.539} C_VEL
LIN {X 0,Y 326.706,Z 246.28,A -85,B 0,C 180,E1 -14921.171,E2 -14921.171} C_VEL
LIN {X 0,Y 326.76,Z 246.276,A -85,B 0,C 180,E1 -14925.429,E2 -14925.429} C_VEL
LIN {X 0,Y 326.752,Z 246.282,A -85,B 0,C 180,E1 -14928.834,E2 -14928.834} C_VEL
LIN {X 0,Y 326.915,Z 246.256,A -85,B 0,C 180,E1 -14932.585,E2 -14932.585} C_VEL
LIN {X 0,Y 326.74,Z 246.283,A -85,B 0,C 180,E1 -14935.06,E2 -14935.06} C_VEL
LIN {X 0,Y 326.992,Z 246.247,A -85,B 0,C 180,E1 -14937.532,E2 -14937.532} C_VEL
LIN {X 0,Y 327.016,Z 246.241,A -85,B 0,C 180,E1 -14941.227,E2 -14941.227} C_VEL
LIN {X 0,Y 326.724,Z 246.288,A -85,B 0,C 180,E1 -14943.696,E2 -14943.696} C_VEL
LIN {X 0,Y 326.906,Z 246.258,A -85,B 0,C 180,E1 -14946.447,E2 -14946.447} C_VEL
LIN {X 0,Y 326.768,Z 246.275,A -85,B 0,C 180,E1 -14949.903,E2 -14949.903} C_VEL
LIN {X 0,Y 326.744,Z 246.279,A -85,B 0,C 180,E1 -14953.681,E2 -14953.681} C_VEL
LIN {X 0,Y 326.647,Z 246.291,A -85,B 0,C 180,E1 -14957.526,E2 -14957.526} C_VEL
LIN {X 0,Y 326.632,Z 246.296,A -85,B 0,C 180,E1 -14960.132,E2 -14960.132} C_VEL
LIN {X 0,Y 326.614,Z 246.302,A -85,B 0,C 180,E1 -14964.126,E2 -14964.126} C_VEL
LIN {X 0,Y 326.582,Z 246.296,A -85,B 0,C 180,E1 -14968.08,E2 -14968.08} C_VEL
LIN {X 0,Y 326.55,Z 246.307,A -85,B 0,C 180,E1 -14971.093,E2 -14971.093} C_VEL
LIN {X 0,Y 326.583,Z 246.306,A -85,B 0,C 180,E1 -14974.016,E2 -14974.016} C_VEL
LIN {X 0,Y 326.633,Z 246.469,A -85,B 0,C 180,E1 -14977.672,E2 -14977.672} C_VEL
LIN {X 0,Y 328.809,Z 255.84,A -85,B 0,C 180,E1 -14980.679,E2 -14980.679} C_VEL
LIN {X 0,Y 329.746,Z 259.998,A -85,B 0,C 180,E1 -14981.865,E2 -14981.865} C_VEL
LIN {X 0,Y 334.821,Z 272.612,A -85,B 0,C 180,E1 -14982.647,E2 -14982.647} C_VEL
LIN {X 0,Y 338.589,Z 292.709,A -85,B 0,C 180,E1 -14983.451,E2 -14983.451} C_VEL
LIN {X 0,Y 336.649,Z 367.562,A -85,B 0,C 180,E1 -14985.11,E2 -14985.11} C_VEL
LIN {X 0,Y 335.886,Z 380.988,A -85,B 0,C 180,E1 -14985.645,E2 -14985.645} C_VEL
LIN {X 0,Y 334.98,Z 393.52,A -85,B 0,C 180,E1 -14986.393,E2 -14986.393} C_VEL
LIN {X 0,Y 333.786,Z 405.553,A -85,B 0,C 180,E1 -14987.372,E2 -14987.372} C_VEL
LIN {X 0,Y 332.332,Z 417.508,A -85,B 0,C 180,E1 -14988.636,E2 -14988.636} C_VEL
LIN {X 0,Y 330.778,Z 428.395,A -85,B 0,C 180,E1 -14990.103,E2 -14990.103} C_VEL
LIN {X 0,Y 329.299,Z 438.158,A -85,B 0,C 180,E1 -14991.764,E2 -14991.764} C_VEL
LIN {X 0,Y 328.102,Z 446.493,A -85,B 0,C 180,E1 -14993.531,E2 -14993.531} C_VEL
LIN {X 0,Y 327.027,Z 453.29,A -85,B 0,C 180,E1 -14995.322,E2 -14995.322} C_VEL
LIN {X 0,Y 326.1,Z 459.481,A -85,B 0,C 180,E1 -14997.4,E2 -14997.4} C_VEL
LIN {X 0,Y 325.657,Z 462.852,A -85,B 0,C 180,E1 -14998.807,E2 -14998.807} C_VEL
LIN {X 0,Y 325.165,Z 466.685,A -85,B 0,C 180,E1 -15000.903,E2 -15000.903} C_VEL
LIN {X 0,Y 324.786,Z 469.244,A -85,B 0,C 180,E1 -15002.974,E2 -15002.974} C_VEL
LIN {X 0,Y 324.574,Z 470.8,A -85,B 0,C 180,E1 -15005.412,E2 -15005.412} C_VEL
LIN {X 0,Y 324.48,Z 470.977,A -85,B 0,C 180,E1 -15007.055,E2 -15007.055} C_VEL
LIN {X 0,Y 324.558,Z 470.532,A -85,B 0,C 180,E1 -15008.594,E2 -15008.594} C_VEL
LIN {X 0,Y 324.606,Z 469.795,A -85,B 0,C 180,E1 -15009.733,E2 -15009.733} C_VEL
LIN {X 0,Y 324.927,Z 467.126,A -85,B 0,C 180,E1 -15012.099,E2 -15012.099} C_VEL
LIN {X 0,Y 325.305,Z 463.191,A -85,B 0,C 180,E1 -15014.334,E2 -15014.334} C_VEL
LIN {X 0,Y 325.849,Z 458.492,A -85,B 0,C 180,E1 -15016.277,E2 -15016.277} C_VEL
LIN {X 0,Y 326.553,Z 452.482,A -85,B 0,C 180,E1 -15018.203,E2 -15018.203} C_VEL
LIN {X 0,Y 327.516,Z 444.929,A -85,B 0,C 180,E1 -15020.116,E2 -15020.116} C_VEL
LIN {X 0,Y 328.546,Z 437.21,A -85,B 0,C 180,E1 -15021.699,E2 -15021.699} C_VEL
LIN {X 0,Y 329.753,Z 427.84,A -85,B 0,C 180,E1 -15023.269,E2 -15023.269} C_VEL
LIN {X 0,Y 331.025,Z 417.378,A -85,B 0,C 180,E1 -15024.671,E2 -15024.671} C_VEL
LIN {X 0,Y 332.285,Z 405.717,A -85,B 0,C 180,E1 -15025.908,E2 -15025.908} C_VEL
LIN {X 0,Y 333.374,Z 393.567,A -85,B 0,C 180,E1 -15026.904,E2 -15026.904} C_VEL
LIN {X 0,Y 334.214,Z 380.835,A -85,B 0,C 180,E1 -15027.666,E2 -15027.666} C_VEL
LIN {X 0,Y 334.921,Z 367.522,A -85,B 0,C 180,E1 -15028.197,E2 -15028.197} C_VEL
LIN {X 0,Y 336.491,Z 290.415,A -85,B 0,C 180,E1 -15029.906,E2 -15029.906} C_VEL
LIN {X 0,Y 331.952,Z 266.81,A -85,B 0,C 180,E1 -15030.762,E2 -15030.762} C_VEL
LIN {X 0,Y 329.648,Z 260.008,A -85,B 0,C 180,E1 -15031.124,E2 -15031.124} C_VEL
LIN {X 0,Y 328.377,Z 253.559,A -85,B 0,C 180,E1 -15033.068,E2 -15033.068} C_VEL
LIN {X 0,Y 326.831,Z 246.411,A -85,B 0,C 180,E1 -15035.399,E2 -15035.399} C_VEL
LIN {X 0,Y 326.924,Z 246.261,A -85,B 0,C 180,E1 -15037.412,E2 -15037.412} C_VEL
LIN {X 0,Y 326.739,Z 246.287,A -85,B 0,C 180,E1 -15041.163,E2 -15041.163} C_VEL
LIN {X 0,Y 326.722,Z 246.286,A -85,B 0,C 180,E1 -15044.96,E2 -15044.96} C_VEL
LIN {X 0,Y 326.702,Z 246.287,A -85,B 0,C 180,E1 -15048.841,E2 -15048.841} C_VEL
LIN {X 0,Y 326.567,Z 246.303,A -85,B 0,C 180,E1 -15052.792,E2 -15052.792} C_VEL
LIN {X 0,Y 326.607,Z 246.297,A -85,B 0,C 180,E1 -15055.492,E2 -15055.492} C_VEL
LIN {X 0,Y 326.571,Z 246.297,A -85,B 0,C 180,E1 -15058.26,E2 -15058.26} C_VEL
LIN {X 0,Y 326.56,Z 246.297,A -85,B 0,C 180,E1 -15060.097,E2 -15060.097} C_VEL
LIN {X 0,Y 325.926,Z 246.385,A -85,B 0,C 180,E1 -15061.126,E2 -15061.126} C_VEL
LIN {X 0,Y 323.125,Z 246.732,A -85,B 0,C 180,E1 -15062.802,E2 -15062.802} C_VEL
LIN {X 0,Y 320.717,Z 247.025,A -85,B 0,C 180,E1 -15064.16,E2 -15064.16} C_VEL
LIN {X 0,Y 319.653,Z 247.15,A -85,B 0,C 180,E1 -15065.211,E2 -15065.211} C_VEL
LIN {X 0,Y 319.551,Z 247.163,A -85,B 0,C 180,E1 -15065.567,E2 -15065.567} C_VEL
LIN {X 0,Y 319.505,Z 247.184,A -85,B 0,C 180,E1 -15069.666,E2 -15069.666} C_VEL
LIN {X 0,Y 319.496,Z 247.172,A -85,B 0,C 180,E1 -15073.464,E2 -15073.464} C_VEL
LIN {X 0,Y 319.53,Z 247.183,A -85,B 0,C 180,E1 -15077.02,E2 -15077.02} C_VEL
LIN {X 0,Y 319.497,Z 247.166,A -85,B 0,C 180,E1 -15080.371,E2 -15080.371} C_VEL
LIN {X 0,Y 319.562,Z 247.172,A -85,B 0,C 180,E1 -15084.463,E2 -15084.463} C_VEL
LIN {X 0,Y 319.51,Z 247.177,A -85,B 0,C 180,E1 -15088.142,E2 -15088.142} C_VEL
LIN {X 0,Y 319.532,Z 247.152,A -85,B 0,C 180,E1 -15091.618,E2 -15091.618} C_VEL
LIN {X 0,Y 319.532,Z 247.179,A -85,B 0,C 180,E1 -15095.304,E2 -15095.304} C_VEL
LIN {X 0,Y 319.558,Z 247.174,A -85,B 0,C 180,E1 -15098.05,E2 -15098.05} C_VEL
LIN {X 0,Y 319.619,Z 247.135,A -85,B 0,C 180,E1 -15102.076,E2 -15102.076} C_VEL
LIN {X 0,Y 319.727,Z 247.152,A -85,B 0,C 180,E1 -15106.012,E2 -15106.012} C_VEL
LIN {X 0,Y 319.732,Z 247.153,A -85,B 0,C 180,E1 -15109.877,E2 -15109.877} C_VEL
LIN {X 0,Y 319.897,Z 247.103,A -85,B 0,C 180,E1 -15113.698,E2 -15113.698} C_VEL
LIN {X 0,Y 319.956,Z 247.119,A -85,B 0,C 180,E1 -15117.486,E2 -15117.486} C_VEL
LIN {X 0,Y 320.013,Z 247.116,A -85,B 0,C 180,E1 -15121.263,E2 -15121.263} C_VEL
LIN {X 0,Y 319.919,Z 247.107,A -85,B 0,C 180,E1 -15126.31,E2 -15126.31} C_VEL
LIN {X 0,Y 319.742,Z 247.155,A -85,B 0,C 180,E1 -15130.132,E2 -15130.132} C_VEL
LIN {X 0,Y 319.739,Z 247.14,A -85,B 0,C 180,E1 -15133.996,E2 -15133.996} C_VEL
LIN {X 0,Y 319.634,Z 247.162,A -85,B 0,C 180,E1 -15137.932,E2 -15137.932} C_VEL
LIN {X 0,Y 319.578,Z 247.17,A -85,B 0,C 180,E1 -15141.957,E2 -15141.957} C_VEL
LIN {X 0,Y 319.581,Z 247.169,A -85,B 0,C 180,E1 -15146.097,E2 -15146.097} C_VEL
LIN {X 0,Y 319.554,Z 247.179,A -85,B 0,C 180,E1 -15148.941,E2 -15148.941} C_VEL
LIN {X 0,Y 319.535,Z 247.169,A -85,B 0,C 180,E1 -15151.865,E2 -15151.865} C_VEL
LIN {X 0,Y 319.592,Z 247.173,A -85,B 0,C 180,E1 -15155.545,E2 -15155.545} C_VEL
LIN {X 0,Y 319.541,Z 247.184,A -85,B 0,C 180,E1 -15159.664,E2 -15159.664} C_VEL
LIN {X 0,Y 319.533,Z 247.176,A -85,B 0,C 180,E1 -15163.462,E2 -15163.462} C_VEL
LIN {X 0,Y 319.564,Z 247.174,A -85,B 0,C 180,E1 -15167.017,E2 -15167.017} C_VEL
LIN {X 0,Y 319.528,Z 247.184,A -85,B 0,C 180,E1 -15170.367,E2 -15170.367} C_VEL
LIN {X 0,Y 319.593,Z 247.176,A -85,B 0,C 180,E1 -15174.458,E2 -15174.458} C_VEL
LIN {X 0,Y 319.545,Z 247.185,A -85,B 0,C 180,E1 -15178.139,E2 -15178.139} C_VEL
LIN {X 0,Y 319.587,Z 247.267,A -85,B 0,C 180,E1 -15179.058,E2 -15179.058} C_VEL
LIN {X 0,Y 321.811,Z 257.525,A -85,B 0,C 180,E1 -15182.349,E2 -15182.349} C_VEL
LIN {X 0,Y 323.624,Z 267.364,A -85,B 0,C 180,E1 -15185.289,E2 -15185.289} C_VEL
LIN {X 0,Y 323.651,Z 268.313,A -85,B 0,C 180,E1 -15185.482,E2 -15185.482} C_VEL
LIN {X 0,Y 327.883,Z 292.55,A -85,B 0,C 180,E1 -15186.399,E2 -15186.399} C_VEL
LIN {X 0,Y 329.787,Z 305.502,A -85,B 0,C 180,E1 -15186.838,E2 -15186.838} C_VEL
LIN {X 0,Y 328.146,Z 376.537,A -85,B 0,C 180,E1 -15188.443,E2 -15188.443} C_VEL
LIN {X 0,Y 327.369,Z 390.242,A -85,B 0,C 180,E1 -15189.006,E2 -15189.006} C_VEL
LIN {X 0,Y 326.391,Z 402.631,A -85,B 0,C 180,E1 -15189.764,E2 -15189.764} C_VEL
LIN {X 0,Y 325.189,Z 414.511,A -85,B 0,C 180,E1 -15190.756,E2 -15190.756} C_VEL
LIN {X 0,Y 323.862,Z 425.942,A -85,B 0,C 180,E1 -15191.986,E2 -15191.986} C_VEL
LIN {X 0,Y 322.598,Z 436.251,A -85,B 0,C 180,E1 -15193.384,E2 -15193.384} C_VEL
LIN {X 0,Y 321.508,Z 444.678,A -85,B 0,C 180,E1 -15194.792,E2 -15194.792} C_VEL
LIN {X 0,Y 320.29,Z 453.811,A -85,B 0,C 180,E1 -15196.679,E2 -15196.679} C_VEL
LIN {X 0,Y 319.288,Z 461.164,A -85,B 0,C 180,E1 -15198.573,E2 -15198.573} C_VEL
LIN {X 0,Y 318.623,Z 467.052,A -85,B 0,C 180,E1 -15200.477,E2 -15200.477} C_VEL
LIN {X 0,Y 318.13,Z 471.678,A -85,B 0,C 180,E1 -15202.382,E2 -15202.382} C_VEL
LIN {X 0,Y 317.877,Z 475.112,A -85,B 0,C 180,E1 -15204.242,E2 -15204.242} C_VEL
LIN {X 0,Y 317.782,Z 477.685,A -85,B 0,C 180,E1 -15206.195,E2 -15206.195} C_VEL
LIN {X 0,Y 317.735,Z 478.828,A -85,B 0,C 180,E1 -15207.463,E2 -15207.463} C_VEL
LIN {X 0,Y 317.697,Z 479.538,A -85,B 0,C 180,E1 -15208.731,E2 -15208.731} C_VEL
LIN {X 0,Y 317.711,Z 479.861,A -85,B 0,C 180,E1 -15209.999,E2 -15209.999} C_VEL
LIN {X 0,Y 317.697,Z 479.796,A -85,B 0,C 180,E1 -15211.267,E2 -15211.267} C_VEL
LIN {X 0,Y 317.736,Z 479.326,A -85,B 0,C 180,E1 -15212.534,E2 -15212.534} C_VEL
LIN {X 0,Y 317.79,Z 478.427,A -85,B 0,C 180,E1 -15213.803,E2 -15213.803} C_VEL
LIN {X 0,Y 317.979,Z 475.438,A -85,B 0,C 180,E1 -15216.344,E2 -15216.344} C_VEL
LIN {X 0,Y 318.308,Z 472.03,A -85,B 0,C 180,E1 -15218.25,E2 -15218.25} C_VEL
LIN {X 0,Y 318.895,Z 467.551,A -85,B 0,C 180,E1 -15220.154,E2 -15220.154} C_VEL
LIN {X 0,Y 319.736,Z 461.876,A -85,B 0,C 180,E1 -15222.052,E2 -15222.052} C_VEL
LIN {X 0,Y 320.879,Z 454.767,A -85,B 0,C 180,E1 -15223.94,E2 -15223.94} C_VEL
LIN {X 0,Y 322.348,Z 445.915,A -85,B 0,C 180,E1 -15225.814,E2 -15225.814} C_VEL
LIN {X 0,Y 323.731,Z 436.155,A -85,B 0,C 180,E1 -15227.483,E2 -15227.483} C_VEL
LIN {X 0,Y 325.087,Z 426.875,A -85,B 0,C 180,E1 -15228.757,E2 -15228.757} C_VEL
LIN {X 0,Y 326.589,Z 415.807,A -85,B 0,C 180,E1 -15229.974,E2 -15229.974} C_VEL
LIN {X 0,Y 327.993,Z 403.434,A -85,B 0,C 180,E1 -15231.032,E2 -15231.032} C_VEL
LIN {X 0,Y 329.098,Z 391.677,A -85,B 0,C 180,E1 -15231.779,E2 -15231.779} C_VEL
LIN {X 0,Y 329.982,Z 378.953,A -85,B 0,C 180,E1 -15232.335,E2 -15232.335} C_VEL
LIN {X 0,Y 330.586,Z 360.122,A -85,B 0,C 180,E1 -15232.817,E2 -15232.817} C_VEL
LIN {X 0,Y 331.913,Z 304.898,A -85,B 0,C 180,E1 -15234.053,E2 -15234.053} C_VEL
LIN {X 0,Y 327.821,Z 281.862,A -85,B 0,C 180,E1 -15234.98,E2 -15234.98} C_VEL
LIN {X 0,Y 325.429,Z 271.375,A -85,B 0,C 180,E1 -15235.462,E2 -15235.462} C_VEL
LIN {X 0,Y 323.993,Z 267.558,A -85,B 0,C 180,E1 -15235.749,E2 -15235.749} C_VEL
LIN {X 0,Y 322.364,Z 259.03,A -85,B 0,C 180,E1 -15238.305,E2 -15238.305} C_VEL
LIN {X 0,Y 320.145,Z 249.61,A -85,B 0,C 180,E1 -15241.357,E2 -15241.357} C_VEL
LIN {X 0,Y 319.575,Z 247.231,A -85,B 0,C 180,E1 -15242.25,E2 -15242.25} C_VEL
LIN {X 0,Y 319.563,Z 247.171,A -85,B 0,C 180,E1 -15246.425,E2 -15246.425} C_VEL
LIN {X 0,Y 319.535,Z 247.172,A -85,B 0,C 180,E1 -15249.659,E2 -15249.659} C_VEL
LIN {X 0,Y 319.525,Z 247.18,A -85,B 0,C 180,E1 -15253.457,E2 -15253.457} C_VEL
LIN {X 0,Y 319.556,Z 247.18,A -85,B 0,C 180,E1 -15257.013,E2 -15257.013} C_VEL
LIN {X 0,Y 319.518,Z 247.185,A -85,B 0,C 180,E1 -15260.363,E2 -15260.363} C_VEL
LIN {X 0,Y 319.581,Z 247.172,A -85,B 0,C 180,E1 -15264.454,E2 -15264.454} C_VEL
LIN {X 0,Y 319.526,Z 247.179,A -85,B 0,C 180,E1 -15268.134,E2 -15268.134} C_VEL
LIN {X 0,Y 319.57,Z 247.174,A -85,B 0,C 180,E1 -15271.601,E2 -15271.601} C_VEL
LIN {X 0,Y 319.572,Z 247.176,A -85,B 0,C 180,E1 -15275.298,E2 -15275.298} C_VEL
LIN {X 0,Y 319.566,Z 247.172,A -85,B 0,C 180,E1 -15278.042,E2 -15278.042} C_VEL
LIN {X 0,Y 319.656,Z 247.159,A -85,B 0,C 180,E1 -15280.975,E2 -15280.975} C_VEL
LIN {X 0,Y 319.709,Z 247.156,A -85,B 0,C 180,E1 -15285.285,E2 -15285.285} C_VEL
LIN {X 0,Y 319.709,Z 247.158,A -85,B 0,C 180,E1 -15288.585,E2 -15288.585} C_VEL
LIN {X 0,Y 319.872,Z 247.133,A -85,B 0,C 180,E1 -15292.421,E2 -15292.421} C_VEL
LIN {X 0,Y 319.711,Z 247.16,A -85,B 0,C 180,E1 -15294.951,E2 -15294.951} C_VEL
LIN {X 0,Y 320.003,Z 247.123,A -85,B 0,C 180,E1 -15298.737,E2 -15298.737} C_VEL
LIN {X 0,Y 319.924,Z 247.131,A -85,B 0,C 180,E1 -15302.514,E2 -15302.514} C_VEL
LIN {X 0,Y 319.872,Z 247.135,A -85,B 0,C 180,E1 -15306.428,E2 -15306.428} C_VEL
LIN {X 0,Y 319.72,Z 247.154,A -85,B 0,C 180,E1 -15310.124,E2 -15310.124} C_VEL
LIN {X 0,Y 319.717,Z 247.155,A -85,B 0,C 180,E1 -15313.988,E2 -15313.988} C_VEL
LIN {X 0,Y 319.608,Z 247.171,A -85,B 0,C 180,E1 -15317.925,E2 -15317.925} C_VEL
LIN {X 0,Y 319.58,Z 247.175,A -85,B 0,C 180,E1 -15320.596,E2 -15320.596} C_VEL
LIN {X 0,Y 319.534,Z 247.179,A -85,B 0,C 180,E1 -15323.317,E2 -15323.317} C_VEL
LIN {X 0,Y 319.551,Z 247.18,A -85,B 0,C 180,E1 -15326.09,E2 -15326.09} C_VEL
LIN {X 0,Y 319.521,Z 247.173,A -85,B 0,C 180,E1 -15328.934,E2 -15328.934} C_VEL
LIN {X 0,Y 319.501,Z 247.179,A -85,B 0,C 180,E1 -15331.859,E2 -15331.859} C_VEL
LIN {X 0,Y 319.555,Z 247.175,A -85,B 0,C 180,E1 -15335.539,E2 -15335.539} C_VEL
LIN {X 0,Y 319.584,Z 247.338,A -85,B 0,C 180,E1 -15337.116,E2 -15337.116} C_VEL
LIN {X 0,Y 321.902,Z 257.189,A -85,B 0,C 180,E1 -15340.365,E2 -15340.365} C_VEL
LIN {X 0,Y 322.531,Z 259.991,A -85,B 0,C 180,E1 -15341.176,E2 -15341.176} C_VEL
LIN {X 0,Y 328.236,Z 273.648,A -85,B 0,C 180,E1 -15342.094,E2 -15342.094} C_VEL
LIN {X 0,Y 330.672,Z 284.726,A -85,B 0,C 180,E1 -15342.586,E2 -15342.586} C_VEL
LIN {X 0,Y 332.175,Z 293.868,A -85,B 0,C 180,E1 -15342.941,E2 -15342.941} C_VEL
LIN {X 0,Y 330.189,Z 367.722,A -85,B 0,C 180,E1 -15344.612,E2 -15344.612} C_VEL
LIN {X 0,Y 329.367,Z 381.484,A -85,B 0,C 180,E1 -15345.175,E2 -15345.175} C_VEL
LIN {X 0,Y 328.422,Z 393.886,A -85,B 0,C 180,E1 -15345.937,E2 -15345.937} C_VEL
LIN {X 0,Y 327.204,Z 405.519,A -85,B 0,C 180,E1 -15346.902,E2 -15346.902} C_VEL
LIN {X 0,Y 325.862,Z 416.257,A -85,B 0,C 180,E1 -15348.044,E2 -15348.044} C_VEL
LIN {X 0,Y 324.288,Z 426.84,A -85,B 0,C 180,E1 -15349.448,E2 -15349.448} C_VEL
LIN {X 0,Y 322.734,Z 436.794,A -85,B 0,C 180,E1 -15351.112,E2 -15351.112} C_VEL
LIN {X 0,Y 321.335,Z 445.868,A -85,B 0,C 180,E1 -15353.027,E2 -15353.027} C_VEL
LIN {X 0,Y 320.269,Z 452.238,A -85,B 0,C 180,E1 -15354.69,E2 -15354.69} C_VEL
LIN {X 0,Y 319.269,Z 458.596,A -85,B 0,C 180,E1 -15356.76,E2 -15356.76} C_VEL
LIN {X 0,Y 318.588,Z 463.342,A -85,B 0,C 180,E1 -15358.777,E2 -15358.777} C_VEL
LIN {X 0,Y 318.076,Z 467.052,A -85,B 0,C 180,E1 -15360.917,E2 -15360.917} C_VEL
LIN {X 0,Y 317.821,Z 468.832,A -85,B 0,C 180,E1 -15362.332,E2 -15362.332} C_VEL
LIN {X 0,Y 317.597,Z 470.087,A -85,B 0,C 180,E1 -15363.733,E2 -15363.733} C_VEL
LIN {X 0,Y 317.481,Z 470.836,A -85,B 0,C 180,E1 -15365.162,E2 -15365.162} C_VEL
LIN {X 0,Y 317.392,Z 471.112,A -85,B 0,C 180,E1 -15366.512,E2 -15366.512} C_VEL
LIN {X 0,Y 317.448,Z 470.706,A -85,B 0,C 180,E1 -15368.393,E2 -15368.393} C_VEL
LIN {X 0,Y 317.613,Z 469.121,A -85,B 0,C 180,E1 -15370.616,E2 -15370.616} C_VEL
LIN {X 0,Y 317.912,Z 466.561,A -85,B 0,C 180,E1 -15372.637,E2 -15372.637} C_VEL
LIN {X 0,Y 318.281,Z 462.922,A -85,B 0,C 180,E1 -15374.636,E2 -15374.636} C_VEL
LIN {X 0,Y 318.869,Z 458.042,A -85,B 0,C 180,E1 -15376.637,E2 -15376.637} C_VEL
LIN {X 0,Y 319.62,Z 451.942,A -85,B 0,C 180,E1 -15378.587,E2 -15378.587} C_VEL
LIN {X 0,Y 320.639,Z 444.499,A -85,B 0,C 180,E1 -15380.482,E2 -15380.482} C_VEL
LIN {X 0,Y 321.732,Z 436.384,A -85,B 0,C 180,E1 -15382.154,E2 -15382.154} C_VEL
LIN {X 0,Y 323.002,Z 426.771,A -85,B 0,C 180,E1 -15383.755,E2 -15383.755} C_VEL
LIN {X 0,Y 324.371,Z 415.557,A -85,B 0,C 180,E1 -15385.241,E2 -15385.241} C_VEL
LIN {X 0,Y 325.693,Z 403.996,A -85,B 0,C 180,E1 -15386.444,E2 -15386.444} C_VEL
LIN {X 0,Y 326.734,Z 392.272,A -85,B 0,C 180,E1 -15387.381,E2 -15387.381} C_VEL
LIN {X 0,Y 327.629,Z 379.029,A -85,B 0,C 180,E1 -15388.157,E2 -15388.157} C_VEL
LIN {X 0,Y 328.32,Z 365.709,A -85,B 0,C 180,E1 -15388.659,E2 -15388.659} C_VEL
LIN {X 0,Y 329.902,Z 291.49,A -85,B 0,C 180,E1 -15390.324,E2 -15390.324} C_VEL
LIN {X 0,Y 325.533,Z 268.798,A -85,B 0,C 180,E1 -15391.171,E2 -15391.171} C_VEL
LIN {X 0,Y 322.534,Z 260.291,A -85,B 0,C 180,E1 -15391.629,E2 -15391.629} C_VEL
LIN {X 0,Y 322.29,Z 259.182,A -85,B 0,C 180,E1 -15391.876,E2 -15391.876} C_VEL
LIN {X 0,Y 319.861,Z 247.206,A -85,B 0,C 180,E1 -15395.833,E2 -15395.833} C_VEL
LIN {X 0,Y 319.804,Z 247.144,A -85,B 0,C 180,E1 -15398.85,E2 -15398.85} C_VEL
LIN {X 0,Y 319.651,Z 247.156,A -85,B 0,C 180,E1 -15402.702,E2 -15402.702} C_VEL
LIN {X 0,Y 319.668,Z 247.167,A -85,B 0,C 180,E1 -15405.298,E2 -15405.298} C_VEL
LIN {X 0,Y 319.62,Z 247.169,A -85,B 0,C 180,E1 -15409.259,E2 -15409.259} C_VEL
LIN {X 0,Y 319.521,Z 247.181,A -85,B 0,C 180,E1 -15413.324,E2 -15413.324} C_VEL
LIN {X 0,Y 319.543,Z 247.182,A -85,B 0,C 180,E1 -15416.097,E2 -15416.097} C_VEL
LIN {X 0,Y 319.504,Z 247.172,A -85,B 0,C 180,E1 -15418.943,E2 -15418.943} C_VEL
LIN {X 0,Y 319.496,Z 247.186,A -85,B 0,C 180,E1 -15421.867,E2 -15421.867} C_VEL
LIN {X 0,Y 319.551,Z 247.163,A -85,B 0,C 180,E1 -15425.567,E2 -15425.567} C_VEL
LIN {X 0,Y 318.836,Z 247.262,A -85,B 0,C 180,E1 -15426.618,E2 -15426.618} C_VEL
LIN {X 0,Y 315.949,Z 247.63,A -85,B 0,C 180,E1 -15428.33,E2 -15428.33} C_VEL
LIN {X 0,Y 313.526,Z 247.929,A -85,B 0,C 180,E1 -15429.717,E2 -15429.717} C_VEL
LIN {X 0,Y 312.488,Z 248.05,A -85,B 0,C 180,E1 -15430.791,E2 -15430.791} C_VEL
LIN {X 0,Y 312.402,Z 248.056,A -85,B 0,C 180,E1 -15431.155,E2 -15431.155} C_VEL
LIN {X 0,Y 312.429,Z 248.055,A -85,B 0,C 180,E1 -15434.215,E2 -15434.215} C_VEL
LIN {X 0,Y 312.434,Z 248.063,A -85,B 0,C 180,E1 -15437.93,E2 -15437.93} C_VEL
LIN {X 0,Y 312.459,Z 248.039,A -85,B 0,C 180,E1 -15441.929,E2 -15441.929} C_VEL
LIN {X 0,Y 312.514,Z 248.049,A -85,B 0,C 180,E1 -15444.225,E2 -15444.225} C_VEL
LIN {X 0,Y 312.488,Z 248.056,A -85,B 0,C 180,E1 -15447.338,E2 -15447.338} C_VEL
LIN {X 0,Y 312.472,Z 248.03,A -85,B 0,C 180,E1 -15451.305,E2 -15451.305} C_VEL
LIN {X 0,Y 312.512,Z 248.048,A -85,B 0,C 180,E1 -15454.71,E2 -15454.71} C_VEL
LIN {X 0,Y 312.532,Z 248.054,A -85,B 0,C 180,E1 -15457.53,E2 -15457.53} C_VEL
LIN {X 0,Y 312.576,Z 248.014,A -85,B 0,C 180,E1 -15461.658,E2 -15461.658} C_VEL
LIN {X 0,Y 312.681,Z 248.024,A -85,B 0,C 180,E1 -15465.691,E2 -15465.691} C_VEL
LIN {X 0,Y 312.682,Z 248.034,A -85,B 0,C 180,E1 -15469.646,E2 -15469.646} C_VEL
LIN {X 0,Y 312.794,Z 247.997,A -85,B 0,C 180,E1 -15472.257,E2 -15472.257} C_VEL
LIN {X 0,Y 312.686,Z 248.003,A -85,B 0,C 180,E1 -15474.846,E2 -15474.846} C_VEL
LIN {X 0,Y 312.969,Z 247.997,A -85,B 0,C 180,E1 -15478.718,E2 -15478.718} C_VEL
LIN {X 0,Y 312.98,Z 247.992,A -85,B 0,C 180,E1 -15481.291,E2 -15481.291} C_VEL
LIN {X 0,Y 312.863,Z 247.986,A -85,B 0,C 180,E1 -15486.453,E2 -15486.453} C_VEL
LIN {X 0,Y 312.757,Z 248.024,A -85,B 0,C 180,E1 -15489.054,E2 -15489.054} C_VEL
LIN {X 0,Y 312.64,Z 248.029,A -85,B 0,C 180,E1 -15492.995,E2 -15492.995} C_VEL
LIN {X 0,Y 312.63,Z 248.016,A -85,B 0,C 180,E1 -15495.654,E2 -15495.654} C_VEL
LIN {X 0,Y 312.57,Z 248.048,A -85,B 0,C 180,E1 -15499.715,E2 -15499.715} C_VEL
LIN {X 0,Y 312.533,Z 248.038,A -85,B 0,C 180,E1 -15502.782,E2 -15502.782} C_VEL
LIN {X 0,Y 312.541,Z 248.046,A -85,B 0,C 180,E1 -15505.911,E2 -15505.911} C_VEL
LIN {X 0,Y 312.507,Z 248.05,A -85,B 0,C 180,E1 -15509.658,E2 -15509.658} C_VEL
LIN {X 0,Y 312.532,Z 248.055,A -85,B 0,C 180,E1 -15513.691,E2 -15513.691} C_VEL
LIN {X 0,Y 312.523,Z 248.045,A -85,B 0,C 180,E1 -15517.39,E2 -15517.39} C_VEL
LIN {X 0,Y 312.454,Z 248.063,A -85,B 0,C 180,E1 -15520.719,E2 -15520.719} C_VEL
LIN {X 0,Y 312.464,Z 248.063,A -85,B 0,C 180,E1 -15524.212,E2 -15524.212} C_VEL
LIN {X 0,Y 312.469,Z 248.064,A -85,B 0,C 180,E1 -15527.926,E2 -15527.926} C_VEL
LIN {X 0,Y 312.49,Z 248.058,A -85,B 0,C 180,E1 -15531.926,E2 -15531.926} C_VEL
LIN {X 0,Y 312.544,Z 248.053,A -85,B 0,C 180,E1 -15534.221,E2 -15534.221} C_VEL
LIN {X 0,Y 312.498,Z 248.063,A -85,B 0,C 180,E1 -15538.087,E2 -15538.087} C_VEL
LIN {X 0,Y 312.529,Z 248.23,A -85,B 0,C 180,E1 -15538.713,E2 -15538.713} C_VEL
LIN {X 0,Y 314.8,Z 258.437,A -85,B 0,C 180,E1 -15542.041,E2 -15542.041} C_VEL
LIN {X 0,Y 316.577,Z 267.962,A -85,B 0,C 180,E1 -15544.919,E2 -15544.919} C_VEL
LIN {X 0,Y 317.373,Z 271.104,A -85,B 0,C 180,E1 -15545.129,E2 -15545.129} C_VEL
LIN {X 0,Y 322.738,Z 302.498,A -85,B 0,C 180,E1 -15546.281,E2 -15546.281} C_VEL
LIN {X 0,Y 323.127,Z 307.465,A -85,B 0,C 180,E1 -15546.428,E2 -15546.428} C_VEL
LIN {X 0,Y 321.46,Z 376.525,A -85,B 0,C 180,E1 -15548.021,E2 -15548.021} C_VEL
LIN {X 0,Y 320.673,Z 390.05,A -85,B 0,C 180,E1 -15548.589,E2 -15548.589} C_VEL
LIN {X 0,Y 319.7,Z 401.921,A -85,B 0,C 180,E1 -15549.322,E2 -15549.322} C_VEL
LIN {X 0,Y 318.461,Z 413.966,A -85,B 0,C 180,E1 -15550.332,E2 -15550.332} C_VEL
LIN {X 0,Y 317.06,Z 425.478,A -85,B 0,C 180,E1 -15551.586,E2 -15551.586} C_VEL
LIN {X 0,Y 315.745,Z 435.861,A -85,B 0,C 180,E1 -15553.013,E2 -15553.013} C_VEL
LIN {X 0,Y 314.38,Z 445.993,A -85,B 0,C 180,E1 -15554.77,E2 -15554.77} C_VEL
LIN {X 0,Y 313.16,Z 454.889,A -85,B 0,C 180,E1 -15556.7,E2 -15556.7} C_VEL
LIN {X 0,Y 312.186,Z 462.006,A -85,B 0,C 180,E1 -15558.639,E2 -15558.639} C_VEL
LIN {X 0,Y 311.398,Z 468.492,A -85,B 0,C 180,E1 -15560.909,E2 -15560.909} C_VEL
LIN {X 0,Y 310.954,Z 472.76,A -85,B 0,C 180,E1 -15562.858,E2 -15562.858} C_VEL
LIN {X 0,Y 310.73,Z 475.951,A -85,B 0,C 180,E1 -15564.808,E2 -15564.808} C_VEL
LIN {X 0,Y 310.698,Z 477.538,A -85,B 0,C 180,E1 -15566.108,E2 -15566.108} C_VEL
LIN {X 0,Y 310.66,Z 478.702,A -85,B 0,C 180,E1 -15567.406,E2 -15567.406} C_VEL
LIN {X 0,Y 310.614,Z 479.424,A -85,B 0,C 180,E1 -15568.702,E2 -15568.702} C_VEL
LIN {X 0,Y 310.625,Z 479.757,A -85,B 0,C 180,E1 -15569.999,E2 -15569.999} C_VEL
LIN {X 0,Y 310.614,Z 479.703,A -85,B 0,C 180,E1 -15571.295,E2 -15571.295} C_VEL
LIN {X 0,Y 310.661,Z 479.252,A -85,B 0,C 180,E1 -15572.592,E2 -15572.592} C_VEL
LIN {X 0,Y 310.706,Z 478.365,A -85,B 0,C 180,E1 -15573.89,E2 -15573.89} C_VEL
LIN {X 0,Y 310.914,Z 475.395,A -85,B 0,C 180,E1 -15576.488,E2 -15576.488} C_VEL
LIN {X 0,Y 311.268,Z 472.01,A -85,B 0,C 180,E1 -15578.438,E2 -15578.438} C_VEL
LIN {X 0,Y 311.902,Z 467.553,A -85,B 0,C 180,E1 -15580.384,E2 -15580.384} C_VEL
LIN {X 0,Y 312.909,Z 460.818,A -85,B 0,C 180,E1 -15582.648,E2 -15582.648} C_VEL
LIN {X 0,Y 314.216,Z 453.488,A -85,B 0,C 180,E1 -15584.573,E2 -15584.573} C_VEL
LIN {X 0,Y 315.509,Z 446.04,A -85,B 0,C 180,E1 -15586.166,E2 -15586.166} C_VEL
LIN {X 0,Y 316.982,Z 436.059,A -85,B 0,C 180,E1 -15587.915,E2 -15587.915} C_VEL
LIN {X 0,Y 318.589,Z 425.871,A -85,B 0,C 180,E1 -15589.322,E2 -15589.322} C_VEL
LIN {X 0,Y 320.173,Z 414.595,A -85,B 0,C 180,E1 -15590.56,E2 -15590.56} C_VEL
LIN {X 0,Y 321.525,Z 402.928,A -85,B 0,C 180,E1 -15591.56,E2 -15591.56} C_VEL
LIN {X 0,Y 322.756,Z 390.231,A -85,B 0,C 180,E1 -15592.356,E2 -15592.356} C_VEL
LIN {X 0,Y 323.643,Z 376.831,A -85,B 0,C 180,E1 -15592.923,E2 -15592.923} C_VEL
LIN {X 0,Y 324.44,Z 349.311,A -85,B 0,C 180,E1 -15593.588,E2 -15593.588} C_VEL
LIN {X 0,Y 325.555,Z 306.049,A -85,B 0,C 180,E1 -15594.574,E2 -15594.574} C_VEL
LIN {X 0,Y 321.733,Z 284.183,A -85,B 0,C 180,E1 -15595.478,E2 -15595.478} C_VEL
LIN {X 0,Y 319.468,Z 274.112,A -85,B 0,C 180,E1 -15595.956,E2 -15595.956} C_VEL
LIN {X 0,Y 316.898,Z 267.572,A -85,B 0,C 180,E1 -15596.42,E2 -15596.42} C_VEL
LIN {X 0,Y 315.42,Z 260.379,A -85,B 0,C 180,E1 -15598.622,E2 -15598.622} C_VEL
LIN {X 0,Y 313.084,Z 250.407,A -85,B 0,C 180,E1 -15601.953,E2 -15601.953} C_VEL
LIN {X 0,Y 312.567,Z 248.111,A -85,B 0,C 180,E1 -15602.829,E2 -15602.829} C_VEL
LIN {X 0,Y 312.541,Z 248.048,A -85,B 0,C 180,E1 -15605.946,E2 -15605.946} C_VEL
LIN {X 0,Y 312.461,Z 248.051,A -85,B 0,C 180,E1 -15610.112,E2 -15610.112} C_VEL
